(* CoDeSys 2.3 library: oscat152.lib *)
(* Libraries: Standard.lib 22.11.04 11:21:12 *)

(* Global variable list: Constants *)
VAR_GLOBAL CONSTANT
	(* Mathematische Konstanten *)
	PI : REAL := 3.14159265358979323846264338327950288;	(* Kreiszahl PI *)
	PI2 : REAL := 6.283185307179586476;							(* PI * 2 *)
	e : REAL := 2.71828182845904523536028747135266249;	(* Eulersche Konstante *)

	(* Physikalische Konstanten *)
	C0 : REAL := 299792458 ;										(* Lichtgeschwindigkeit in m/s *)
	EL : REAL := 1.60217653E-19;									(* elementarladung in Colomb = A * s *)
	GN : REAL := 9.80665; 											(* Erdbeschleunigung in m / s² *)
	TK : REAL := -273.15;												(* absoluter Nullpunkt in °C *)

END_VAR

VAR_GLOBAL
END_VAR

(* revisionhistory
hm 3.3.2007
	extended accuracy of pi2
	renamed T0 to Tk for better compatibility with other libraries
	renamed C t0 c0 for better compatibility
*)

(* Data type *)
TYPE esr_data :
STRUCT
	typ : BYTE;
	adress : STRING(10);
	DS : DT;
	TS : TIME;
	data : ARRAY[0..7] OF BYTE;
END_STRUCT
END_TYPE

(* POU _array_init, ST *)
FUNCTION _array_init : BOOL
VAR_INPUT
	pt : POINTER TO ARRAY[0..32000] OF REAL;
	size : INT;
	init : REAL;
END_VAR
VAR
	i: INT;
	stop: INT;
END_VAR


(*
version 1.1	9 jan 2007
programmer 	hugo
tested by		tobias

this function will initialize a given array with a value init.
the function needs to be called:	_array_init(adr("array"),sizeof("array"));
this function will manipulate a given array.
the function manipulates the original array, it rerturnes true when finished.
because this function works with pointers its very time efficient and it needs no extra memory.

*)
stop := (size - SIZEOF(pt)) / SIZEOF(pt);
FOR i := 0 TO stop DO
	pt^[i] := init;
END_FOR;
_array_init := TRUE;

(* revision History

hm 6.1.2007	rev 1.1
change typ of function to bool
added _array_init := true to set output true.

*)
END_FUNCTION

(* POU _array_median, ST *)
FUNCTION _array_median : REAL
VAR_INPUT
	pt : POINTER TO ARRAY[0..32000] OF REAL;
	size : INT;
END_VAR
VAR
	i: INT;
	m: INT;
	temp : REAL;
	stop: INT;
END_VAR

(*
version 1.1	3 mar 2007
programmer 	hugo
tested by		tobias

this function will calculate the median of a given array.
in order to do so the ariginal array is sorted and stays sorted after the function finishes
the function needs to be called:	_array_median(adr("array"),sizeof("array"));
this function will manipulate a given array.
the function will return the median of the original array.
for example [12,0,4,7,1] the median is 4 and the array after the function is called is [0,1,4,7,12]
because this function works with pointers its very time efficient and it needs no extra memory.

*)
stop := (size - SIZEOF(pt)) / SIZEOF(pt);
FOR i := 0 TO stop - 1 DO
	FOR m := i + 1 TO stop DO
		IF pt^[i] > pt^[m] THEN
			temp := pt^[i];
			pt^[i] := pt^[m];
			pt^[m] := temp;
		END_IF;
	END_FOR;
END_FOR;
IF even(stop) THEN
	_array_median := pt^[stop/2];
ELSE
	i := stop/2;
	_array_median := (pt^[i] + pt^[i+1])/2;
END_IF;

(* revision history
hm 3.3.2007	rev 1.1
	corrected an error, changed the statement line 14	i := TRUNC(stop/2); to i := stop/2;

*)
END_FUNCTION

(* POU even, ST *)
FUNCTION even : BOOL
VAR_INPUT
	in : INT;
END_VAR
VAR
END_VAR


(*
version 1.0	1 oct 2006
programmer 	hugo
tested by		tobias

this function chacks an input for even  value
the output is true if the input is even.
execution time on wago 750 - 841 =  10  us
*)
IF (in MOD 2) = 0 THEN  even := TRUE; ELSE even := FALSE; END_IF;
END_FUNCTION

(* POU _array_sort, ST *)
FUNCTION _array_sort : BOOL
VAR_INPUT
	pt : POINTER TO ARRAY[0..32000] OF REAL;
	size : INT;
END_VAR
VAR
	i: INT;
	m: INT;
	temp : REAL;
	stop: INT;
END_VAR

(*
version 1.1	6 jan 2007
programmer 	hugo
tested by		tobias

this function will sort a given array.
the function needs to be called:	_array_sort(adr("array"),sizeof("array"));
this function will manipulate a given array.
the function will not return anything except true, it will instead manipulate the original array.
because this function works with pointers its very time efficient and it needs no extra memory.

*)
stop := (size - SIZEOF(pt)) / SIZEOF(pt);
FOR i := 0 TO stop - 1 DO
	FOR m := i + 1 TO stop DO
		IF pt^[i] > pt^[m] THEN
			temp := pt^[i];
			pt^[i] := pt^[m];
			pt^[m] := temp;
		END_IF;
	END_FOR;
END_FOR;
_array_sort := TRUE;

(* revision history

hm 6.1.2007 	rev 1.1
	changed return value to true

*)
END_FUNCTION

(* POU acosH, ST *)
FUNCTION acosH : REAL
VAR_INPUT
	X : REAL;
END_VAR
VAR
END_VAR


(*
version 1.0	12 jan 2007
programmer 	hugo
tested by		tobias

this function calculates the arcus cos hyperbolicus

*)
acosH := LN(X + SQRT(EXPT(x,2)-1));
END_FUNCTION

(* POU acotH, ST *)
FUNCTION acotH : REAL
VAR_INPUT
	X : REAL;
END_VAR
VAR
END_VAR


(*
version 1.0	12 jan 2007
programmer 	hugo
tested by		tobias

this function calculates the arcus cotangens hyperbolicus

*)
acotH := LN((x+1)/(x-1))/2;
END_FUNCTION

(* POU actuator_2P, ST *)
FUNCTION_BLOCK actuator_2P
VAR_INPUT
	val : REAL;
	force : BOOL;
	force_in : BOOL;
END_VAR
VAR_INPUT CONSTANT
	self_act_time : TIME := t#10d;
	self_act_cycles : INT := 5;
	cycle_time : TIME := t#10m;
	min_ontime : TIME := t#10s;
	min_offtime : TIME := t#10s;
END_VAR
VAR_OUTPUT
	out :BOOL;
	pos : REAL;
END_VAR
VAR
	last_activation : TIME;
	count : INT;
	TON : TIME;
END_VAR


(*
version 1.2	17 jan 2007
programmer 	hugo
tested by		tobias

this is an intelligent actuator interface for any 2point actuator like coil drive.
the 2Point actuator can only switch on/off and therefore a input must be converted to on/off cycles.
the interface can be programmed with double click on the symbol for duty cyle, min_ontime and min_offtime to avoid flickering of the valve or flap.
in addition a self_act_time and self_act_cycles ca be programmed to switch n times on/off every self_act_time to avoid a valve to freeze.
a on and off input can be used to force the valve on or off at all times.
a additional pos output will always indicate the current position of a valve.
the input value must be between 0 and 1.

val		force	force_in	pos	out			
X		0		-			X		duty cycle X
-		1		1			1		1
-		1		0			0		0

*)
(* verify input to be between 0 and 1 *)
IF val <0 THEN val := 0; ELSIF val > 1 THEN val := 1; END_IF;

(* check for min ontime or min offtime and wait if not passed *)
IF (out AND TIME() - last_activation < min_ontime) OR (NOT out AND TIME() - last_activation < min_offtime) THEN RETURN;

(* when force off then shutoff valve *)
ELSIF force AND NOT force_in THEN
	pos := 0;
	out := 0;
	last_activation := TIME();
	count := 0;

(* if force on then turn on valve *)

ELSIF force AND force_in THEN
	pos := 1;
	out := 1;
	last_activation := TIME();
	count := 0;

(* if nothing happened for self_act_time then do self activation cycles *)
ELSIF (TIME() - last_activation >= self_act_time AND count = 0 AND self_act_cycles > 0) OR (count > 0 AND count < self_act_cycles * 2) THEN
	out := NOT out;
	last_activation := TIME();
	count := count + 1;
	RETURN;
ELSIF count > 0 THEN
	count := 0;
ELSE
	ton := multime(cycle_time,val);
	IF ton < min_ontime / 2 THEN ton := t#0s; ELSIF ton < min_ontime THEN ton := min_ontime; END_IF;
	IF ton > cycle_time - min_offtime / 2 THEN ton := cycle_time; ELSIF ton > cycle_time - min_offtime THEN ton := cycle_time - min_offtime; END_IF;
	IF ton = t#0s THEN
		IF out =0 THEN
			pos := 0;
			RETURN;
		ELSE
			out := 0;
			pos := 0;
			last_activation := TIME();
		END_IF;
	ELSIF ton = cycle_time THEN
		IF out = 1 THEN
			pos := 1;
			RETURN;
		ELSE
			out := 1;
			pos := 1;
			last_activation := TIME();
		END_IF;
	END_IF;
	pos := TIME_TO_REAL(ton) / TIME_TO_REAL(cycle_time);
	(* output pulse generation *)
	IF out AND TIME() - last_activation >= ton THEN
		out := 0;
		last_activation := TIME();
	ELSIF NOT out AND TIME() - last_activation >= cycle_time - ton THEN
		out := 1;
		last_activation := TIME();
	END_IF;
END_IF;


(*
revision history:

7.10.2006: rev 1.1
	changed error pos could not reach 1 or 0 under certain conditions due to error in code.
	changes on and off in the be force and force_in for better usability.

17.1.2007	rev 1.2
	deleted unused variable time_overflow
*)
END_FUNCTION_BLOCK

(* POU cycle_time, ST *)
FUNCTION_BLOCK cycle_time
VAR_INPUT
	rst : BOOL;
END_VAR
VAR_OUTPUT
	ct_min : TIME := t#0s;
	ct_max : TIME := t#0s;
	ct_last : TIME;
	systime : TIME;
	sysdays : INT;
	cycles : DWORD;
END_VAR
VAR
	last_cycle : TIME;
	tx: TIME;
	init: BOOL;
END_VAR


(*
	version 1.2	10 Mar 2007
	programmer 	hugo
	tested BY		hans

this function block measures the cycle time and displays the last, min and max cycle time of the current task.
the resolution is 1ms.
the cycles output is a dword counter which counts the cycles.
a rst pulse on the input will reset all data.


*)
tx :=TIME() - last_cycle;
IF rst THEN
	ct_min := t#10h;
	ct_max := t#0ms;
	cycles := 0;
ELSIF last_cycle > t#0s THEN
	IF tx < ct_min THEN ct_min := tx;
	ELSIF tx > ct_max THEN ct_max := tx;
	END_IF;
	ct_last := tx;
ELSIF ct_min = t#0s THEN
	ct_min := t#0s - t#1ms;
END_IF;
IF init THEN
	systime := systime + tx;
		IF systime >= t#1d THEN
			systime := systime - t#1d;
			sysdays := sysdays + 1;
		END_IF;
END_IF;
init := TRUE;
last_cycle := last_cycle + tx;
cycles := cycles + 1;

(*	revision history
hm 12.12.2006		rev 1.1
	added cycles output, a dword cycle counter.
hm 10.3.2007			rev 1.2
	changed initialization of ct_min to t#10h for compatibility with siemens s7

*)
END_FUNCTION_BLOCK

(* POU multime, ST *)
FUNCTION multime : TIME
VAR_INPUT
	t : TIME;
	M : REAL;
END_VAR
VAR
END_VAR


(*
version 1.0	2 oct 2006
programmer 	hugo
tested by		tobias

multiplies a time by a real number and returns a time
*)
multime := REAL_TO_TIME(TIME_TO_REAL(t)*M);
END_FUNCTION

(* POU actuator_3P, ST *)
FUNCTION_BLOCK actuator_3P
VAR_INPUT
	in : REAL;
	force : BOOL;
	on : BOOL;
	end_pos : BOOL;
	diag : BOOL;
END_VAR
VAR_INPUT CONSTANT
	min_ontime : TIME := t#10s;
	min_offtime : TIME := t#10s;
	max_runtime : TIME := t#60s;
	auto_diag_time : TIME := t#10d;
	cal_runtime : TIME := t#600s;
	switch_available: BOOL;
END_VAR
VAR_OUTPUT
	out1 : BOOL;
	out2 : BOOL;
	pos : REAL;
	busy : BOOL;
	error : BOOL;
END_VAR
VAR
	val: REAL;
	tx : TIME;
	last_diag: TIME;
	last : TIME;
	runtime_1 : TIME;
	runtime_2 : TIME;
	state : INT;
	rout: FT_rmp;
	end : R_TRIG;
	cal_timer: TIME;
END_VAR


(*
version 1.2	23 Jan 2007
programmer 	hugo
tested by		tobias

actuator_3P is an interface for a 3 point actuator.
a 3P actuator is a motor with 2 directions that drives a valve or flap. the position of the valve or flap is controlled by runtime of the motor foreward or backward.
the available inputs are:
in is a real value which specifies the position of the actuator, 0 = 0% and 1 = 100% any value <0 or > 1 is limited to 0 or 1.
a force input must be low for normal operation and if switched high, the motor can only be controlled for 0% or 100% positions with the on input.
an and pos input is available for a end_pos switch, this switch indicates the valve or flap to be at either 0% or 100%
a diag input can at any time start a diag cycle which turns the motor towards the 0% position, then measures the runtime to 100% and then the runtime to 0%
these runtimes are stored and used for absolute positioning of the motor during normal operation.
a setup constand "auto_diag_time can be used to specify how often the actuator repeates this auto_diag cycla automatically.
at power on a cycle is perfomed automatically.
a 0 for this value means auto diag is never performed.

the outputs ar out1 and out2 for up and down direction of the motor. to avoid flickering the output can be programmed for min_ontime and min_offtime.
a pos outout indicates the absulute position of the actuator during operation and a busy output indicates the actuator is busy.
a error output is initiated when the specified max_runtime is reached by any direction during debug.
also when the up and down direction differs by more then 10% the error output is set.

for absolute positioning accuracy the actuator has a setup variable "cal_runtime" if this is set the actuator measures the total runtime of the motors and when this 
cal_runtime is exceeded it resets the actuator to 0% position and sets the output again to assure absolute accuracy.

autodiag and calibration can be shut off by setting the appropriate values to 0.
a switch_available setup variable specifies if end_pos switches are available.

*)
(* setup *)
tx := TIME() - last;
end(clk := end_pos);

(* init only when first started *)
IF state = 0 THEN
	runtime_1 := max_runtime;
	runtime_2 := max_runtime;
	state := 1;
	rout(KR := 1000 / TIME_TO_REAL(runtime_1), KF := 1000 / TIME_TO_REAL(runtime_1) );
	tx := t#0s;
	last := TIME();
	last_diag := last;
END_IF;

(* check for end_sw and stop if reached *)
IF switch_available AND out1 AND end.Q THEN
	(* upper limit has been reached *)
	out1 := 0;
	rout(rmp := 0, in := 1);
	rout.Rmp := 1;
ELSIF switch_available AND out2 AND end.Q THEN
	(* lower limit has been reached *)
	out2 := 0;
	rout(rmp := 0, in := 0);
	rout.Rmp := 1;
END_IF;

(* check for min_offtime and min_ontime and return if it has not elapsed *)
IF NOT busy AND tx < min_offtime THEN RETURN;
ELSIF busy AND tx < min_ontime THEN RETURN;

(* check for last diag cycle and start diag if auto_diag_time has elapsed *)
ELSIF (tx + last - last_diag > auto_diag_time AND state > 10 AND auto_diag_time > t#0s) OR (diag AND state >= 10) THEN state := 1;

(* check if force pin is high *)
ELSIF force THEN state := 10;

(* check if calibration is necessary *)
ELSIF cal_timer > cal_runtime AND state = 99 AND cal_runtime > t#0s THEN state := 20;
END_IF;

(* state machine for operation *)
CASE state OF

1 :	(* diagnostic start *)
	(* all data is reset and out2 is turned on to make sure we start from top position *)
	last_diag := tx + last;
	diag := 0;
	state := 2;
	pos := 0;
	busy := 1;
	last := tx + last;
	out1 := 0;
	out2 := 1;
	RETURN;

2:	(* wait for max_runtime or end_pos to be reached *)
	IF tx < max_runtime AND NOT end.Q THEN RETURN; END_IF;
	state := 3;
	last := tx + last;
	out1 := 1;
	out2 := 0;
	RETURN;

3: 	(* measure runtime_2 *)
	IF tx < max_runtime AND NOT end.Q THEN RETURN; END_IF;
	state := 4;
	runtime_1 := tx;
	last := tx + last;
	out1 := 0;
	out2 := 1;
	RETURN;

4:	(* measure runtime_1 *)
	IF tx < max_runtime AND NOT end.Q THEN RETURN; END_IF;
	state := 99;
	runtime_2 := tx;
	last := tx + last;
	out2 := 0;
	busy := 0;
	(* reset the output ramp generator to the 0% position as the valve is after diags *)
	rout(rmp := 0, in := 0);
	rout.Rmp := 1;
	cal_timer := t#0s;
	IF differ(TIME_TO_REAL(runtime_1), TIME_TO_REAL(runtime_2), TIME_TO_REAL(max_runtime) * 0.1) THEN error := TRUE;
	ELSIF runtime_1 > multime(max_runtime, 0.9) AND switch_available THEN error := TRUE;
	ELSIF runtime_2 > multime(max_runtime, 0.9) AND switch_available THEN error := TRUE;
	END_IF;
	RETURN;

10: (* force pin is active, outputs are forced on or off by the on pin *)
	IF on AND NOT out2 THEN val := 1;
	ELSIF NOT on AND NOT out1 THEN val := 0;
	END_IF;
	IF NOT force THEN state := 99; END_IF;

20 : (* calibrate to allow for correction of positioning error addig up *)
	cal_timer := t#0s;
	state := 21;
	pos := 0;
	busy := 1;
	last := tx + last;
	out1 := 0;
	out2 := 1;
	RETURN;

21:	(* after end_sw or max_runtime we can be sure to have reached the 0% position *)
	IF tx < max_runtime AND NOT end.Q THEN RETURN; END_IF;
	state := 99;
	out2 := 0;
	busy := 0;
	last := tx + last;
	rout(rmp := 0, in := 0);
	rout.Rmp := 1;
	RETURN;

99: (* normal operation *)
	(* only if input changes for an equivalent of min_ontime then change the output *)
	(* if there is a directional change then wait until last step is finished *)
	IF in < TIME_TO_REAL(min_ontime)/TIME_TO_REAL(max_runtime)/2 THEN val := 0;
	ELSIF in > 1 - TIME_TO_REAL(min_ontime)/TIME_TO_REAL(max_runtime)/2 THEN val := 1;
	ELSIF differ(LIMIT(0,in,1), val, TIME_TO_REAL(min_ontime) / TIME_TO_REAL(max_runtime)) OR in = 0 OR in = 1 THEN
		IF in < val AND NOT out1 THEN val := in;
		ELSIF in > val AND NOT out2 THEN val := in;
		END_IF;
	END_IF;

END_CASE;

(* output ramp generator *)
rout(in := val);
out1 := rout.busy AND rout.UD;
out2 := rout.busy AND NOT rout.UD;
pos := rout.out;

(* set the busy output and if busy goes low, then set the last time in order to check for min_offtime *)
IF NOT busy AND rout.busy THEN
	last := tx + last;
ELSIF busy AND NOT rout.busy THEN
	cal_timer := cal_timer + tx;
	last := tx + last;
END_IF;
busy := rout.busy;



(* revision history

19.10.2006	rev 1.1
	added security checks for end_switch to avoid overrun of the end_switch, hans

23.1.2007		rev 1.2
	deleted unused variables force_on and force_off


*)
END_FUNCTION_BLOCK

(* POU FT_rmp, ST *)
FUNCTION_BLOCK FT_rmp
VAR_INPUT
	Rmp : BOOL := TRUE;
	in : REAL;
	KR : REAL;
	KF : REAL;
END_VAR
VAR_OUTPUT
	out : REAL;
	busy : BOOL;
	UD : BOOL;
END_VAR
VAR
	tx: TIME;
	last: TIME;
	init: BOOL;
END_VAR

(*
	version 1.2	12 Feb 2007
	programmer 	oscat
	tested BY		oscat

this ramp function follows an input signal with a linear ramp up or down, the up or down speed can be set with KF and KR.
a K factor of 1 means 1 unit per second on the output. K factors can only be positive and not negative.
a busy output signals the ramp is running or busy false means the in value is present on the output.
a rmp input false means the output follows the input dierctly while a rmp = true means the output follows the input with a ramp.
a updn output signal the directon of the ramp (up or down).

*)
tx := TIME() - last;
IF NOT init THEN
	init := TRUE;
	last := tx;
	tx := t#0s;
	out := in;
END_IF;
IF NOT rmp THEN
	out := in;
	busy := FALSE;
ELSIF out > in AND kf > 0 THEN
	(* ramp down *)
	out := out - TIME_TO_REAL(tx) / 1000 * KF;
	IF out < in THEN out := in; END_IF;
ELSIF out < in AND kr > 0 THEN
	(* ramp up *)
	out := out + TIME_TO_REAL(tx) / 1000 * KR;
	IF out > in THEN out := in; END_IF;
END_IF;

(* set busy and dir flags *)
IF out < in THEN
	busy := TRUE;
	ud := 1;
ELSIF out > in THEN
	busy := TRUE;
	ud := 0;
ELSE
	busy := FALSE;
END_IF;
last := last + tx;


(* revision history:

hm 8.10.2006			rev 1.1
	added ud output

hm 12. feb 2007		rev 1.12
	added init variable and corrected a possible startup problem
*)
END_FUNCTION_BLOCK

(* POU differ, ST *)
FUNCTION differ : BOOL
VAR_INPUT
	in1 : REAL;
	in2 : REAL;
	X : REAL;
END_VAR
VAR
END_VAR

(*
version 1.0	8 oct 2006
programmer 	hugo
tested by		tobias

this function checks if in1 differs more then x from in2
the output is true if in1 < in2 - x or in1 > in2 + X
*)
differ := in1 < in2 - X OR in1 > in2 + X;
END_FUNCTION

(* POU actuator_pump, ST *)
FUNCTION_BLOCK actuator_pump
VAR_INPUT
	in : BOOL;
	manual : BOOL;
	rst : BOOL := FALSE;
END_VAR
VAR_INPUT CONSTANT
	min_ontime : TIME := t#10s;
	min_offtime : TIME := t#10s;
	run_every : TIME := t#10000m;
END_VAR
VAR_OUTPUT
	pump : BOOL;
	runtime : REAL;
	cycles : REAL;
END_VAR
VAR
	tx : TIME;
	last_change : TIME;
	meter : ontime;
	old_man : BOOL;
	init: BOOL;
END_VAR

(*
	version 1.1	27 dec 2006
	programmer 	oscat
	tested BY		oscat

actuator_pump is a pump interface which can be controlled by an input in and an input manual.
in or manual high turns the pump output on.
a rst input is used to reset the runtime counters.
when the pump was not active for a time run_every the actuator turns on the pump automatically for min_ontime.
two setup variables min_ontime and min_offtime guarantee a minimum runtime and offtime of the pump.
the units are hours and the output type is real to prevent from overfow.

*)
tx := TIME();

IF NOT init THEN
	init := 1;
	last_change := tx;
ELSIF rst THEN
	rst := FALSE;
	meter(rst := 1);
	meter.rst := 0;
ELSIF manual AND NOT pump AND NOT old_man THEN
	last_change := tx;
	pump := 1;
ELSIF NOT manual AND old_man AND pump AND NOT in THEN
	last_change := tx;
	pump := 0;
ELSIF in AND NOT pump AND tx - last_change >= min_offtime THEN
	last_change := tx;
	pump := 1;
ELSIF pump AND NOT in AND NOT manual AND tx - last_change >= min_ontime THEN
	last_change := tx;
	pump := 0;
ELSIF NOT pump AND tx - last_change >= run_every THEN
	last_change := tx;
	pump := 1;
END_IF;

meter(in := pump);
runtime := meter.ontime;
cycles := meter.cycles;
old_man := manual;

(*
27.12.2006	rev 1.1	hm
fixed a failure while the pump would run for tmin after startup.


*)
END_FUNCTION_BLOCK

(* POU ontime, ST *)
FUNCTION_BLOCK ontime
VAR_INPUT
	in : BOOL;
	rst : BOOL := FALSE;
END_VAR
VAR_OUTPUT RETAIN
	ontime : REAL;
	last_on : REAL;
	cycles : REAL;
END_VAR
VAR
	tx: TIME;
	last : TIME;
	power : BOOL := FALSE;
	edge : BOOL := 0;
END_VAR

(*
version 1.1	22 feb 2007
programmer 	oscat
tested by		tobias

M_runtime measures the ontime of a signal in hours.
the output is of type real because the time type will overflow within 49 days.
the units are hours.

*)
(* at first we need to determine if the sps was powered off *)

tx := TIME();
IF NOT power THEN
	power := TRUE;
	cycles := cycles +1;
ELSIF rst THEN
	ontime := 0;
	cycles := 0;
	last_on := 0;
ELSIF in THEN
	ontime := ontime + DWORD_TO_REAL( TIME_TO_DWORD(tx - last))/3600000.0;
	last_on := last_on + DWORD_TO_REAL(TIME_TO_DWORD(tx - last))/3600000.0;
	IF in AND NOT edge THEN
		cycles := cycles +1;
		last_on := 0;
	END_IF;
END_IF;
last := tx;
edge := in;

(* revision history
hm 22.2.2007		rev 1.1
	changed VAR RETAIN PERSISTENT to VAR RETAIN for better compatibility
	wago lon contollers do not support persisitent

*)
END_FUNCTION_BLOCK

(* POU actuator_UD, ST *)
FUNCTION_BLOCK actuator_UD
VAR_INPUT
	UD : BOOL;
	ON : BOOL;
	Manual : BOOL := 0;
	Up : BOOL;
	Dn : BOOL;
	off : BOOL := 0;
	YUP_in : BOOL;
	YDN_in : BOOL;
END_VAR
VAR_INPUT CONSTANT
	TON : TIME;
	TOFF : TIME;
	out_return : BOOL;
END_VAR
VAR_OUTPUT
	Yup : BOOL;
	Ydn : BOOL;
	status : BYTE;
END_VAR
VAR
	tx : TIME;
	last : TIME;
	init: BOOL;
END_VAR

(*
version 1.1	22 jan 2007
programmer 	hugo
tested by		tobias

out_ud is a up/dn or Right/left locked output driver.
it can be controlled by automatic inputs UD and ON as well as manual inputs for up and dn.
a security input to shut off at any time is prvided by the off input.
two time set inputs ton and toff specify a minimum on time for outputs and a minimum off time before the next output can become active.
the module assures that only one output can be active at any time.
for higher security pls make sure you use hardware locking of the outputs to prevent from defective wiring or outputs.
further security is provided b feedback inputs Yup_in and Ydn_in which are separate inputs for the output signal, if these inputs are not available 
pls connect them directly to Yup and Ydn.
manual mode will override automatic mode by setting the manual input high.
a status output will be 0 for normal operation or 1 - 99 for error reporting and 101 - 199 for status reporting
The status output is ESR comptible.
*)
(* read system time *)
tx := TIME();

IF NOT init THEN
	(* INITIALIZATION AT FIRST CALL *)
	last := tx;
	init := TRUE;
ELSIF off THEN
	(* emergency shut off detected *)
	Yup := FALSE;
	Ydn := FALSE;
	last := tx;
	status := 101;

(* WATH FOR MIN TON TIME *)
ELSIF ((Yup OR Ydn) AND tx - last < Ton) THEN RETURN;
ELSIF NOT yup AND NOT ydn AND tx - last < toff THEN	RETURN;

(* manual operation *)
ELSIF manual THEN
	status := 102;
	(* directional chage set both outs 0 first *)
	IF yup AND NOT up OR ydn AND NOT dn THEN
		ydn := 0;
		yup := 0;
		last := tx;
	(* manual up operation *)
	ELSIF UP AND NOT DN AND NOT OFF THEN
		Ydn := 0;
		Yup := 1;
		last := tx;
		status := 103;
	(* manual down operation *)
	ELSIF DN AND NOT UP AND NOT OFF THEN
		Yup := 0;
		Ydn := 1;
		last := tx;
		status := 104;
	(* maual mode but no up or down *)
	ELSE
		IF YUP OR YDN THEN LAST := tx; END_IF;
		Yup := 0;
		Ydn := 0;
	END_IF;

(* automatic operation *)
ELSE
	(* directional change set outputs low first *)
	IF yup AND NOT ud OR ydn AND UD THEN
		yup := 0;
		ydn := 0;
		last := tx;
	(* automatic up operation *)
	ELSIF Ud AND on AND NOT OFF THEN
		Ydn := 0;
		Yup := 1;
		last := tx;
		status := 111;

	(* automatic down operation *)
	ELSIF NOT UD AND on AND NOT OFF THEN
		Yup := 0;
		Ydn := 1;
		last := tx;
		status := 112;
	(* standby mode *)
	ELSE
		IF Yup OR Ydn THEN last := tx; END_IF;
		Yup := 0;
		Ydn := 0;
		status := 110;
	END_IF;
END_IF;

(* make sure Yup and Ydn are never on at the same time *)
IF Ydn AND Yup_in AND out_return THEN
	Ydn := 0;
	status := 1;
END_IF;
IF Yup AND Ydn_in AND out_return THEN
	Yup := 0;
	status := 2;
END_IF;

(* revision history
hm 22. jan 2007	rev 1.1
	added status output
	changed inputs ton, toff to config variables
	added config var out_return to enable yup_in and Ydn_in
	manual mod will override automatic mode 
*)
END_FUNCTION_BLOCK

(* POU AIN, ST *)
FUNCTION AIN : REAL
VAR_INPUT
	in : DWORD;
END_VAR
VAR_INPUT CONSTANT
	Bits : BYTE;
	sign : BYTE := 255;
	low : REAL := 0;
	high : REAL := 10;
END_VAR
VAR
	temp1 : DWORD;
	temp2 : DWORD;
	sx : BOOL;
END_VAR

(*
version 1.2	19 jan 2007
programmer 	oscat
tested by		tobias

Ain converts signals from A/D converters or other analog sources to an internal real value
the lowest number of bits are extracted from the input word and the sign will be extracted if available separately.
the output signal is then conditioned to range from low to high values for a 0 to max value on the analog inputs:
for example a 15bit input (bits := 12) with sign at bit 15 (0..15) will deliver 0.0 (low value at 0) for an input value of 2#0000_0000_0000
an input value of 2#1111_1111_1111 will deliver 10.0 on the output (high value set to 10).

*) 
(* extract the sign bit *)
IF sign < 32 THEN
	temp1 := SHR(in,sign);
	sx := temp1.0;
ELSE
	sx := FALSE;
END_IF;
temp1 := SHR(16#FFFFFFFF,32-bits);
temp2 := in AND temp1;
AIN := (high - low)*temp2 / temp1 + low;
IF sx THEN AIN := AIN * -1; END_IF;

(* revision history
hm 18.8.2006	rev 1.1
	fixed an error with low value negative and high value 0.

hm 19.1.2007	rev 1.2
	fixed an error with sign bit.
*)
END_FUNCTION

(* POU Aout, ST *)
FUNCTION Aout : DWORD
VAR_INPUT
	in : REAL;
END_VAR
VAR_INPUT CONSTANT
	Bits : BYTE;
	sign : BYTE := 255;
	low : REAL := 0;
	high : REAL := 10;
END_VAR
VAR
	in2 : REAL;
	sx : BOOL;
END_VAR

(*
version 1.1	18 jan 2007
programmer 	oscat
tested by		tobias

this module conditions an internal real value for a signal output D/A converter.
Aout converts and internal real value to a word for an D/A converter or other output devices.
The input value is converted to a n-bit wide output and a sign bit is set separately as specified.
the outout min value is set for the specified min input value and the max output is set for the max input value.
an input higher or lower then the max or min value will set the respective max or min value or the output.


*) 
(* if sign bit is defined *)
IF sign < 32 THEN
	sx := sign_R(in);
	in2 := ABS(in);
ELSE
	in2 := in;
END_IF;

(* begrenze in auf die zulässigen werte *)
IF in2 < low THEN
	in2 := low;
ELSIF in2 > high THEN
	in2 := high;
END_IF;

(* Berechne den Ausgnagswert *)
Aout := REAL_TO_DWORD((in2 - low) / (high - low) * (EXPT(2,bits) -1));
IF sx THEN Aout := SHL(2#1,sign) OR Aout; END_IF;

(*
revision history

hm 17.1.2007		rev 1.1
	renamed Modul to aout.
	changed Output to 32 Bit max.
	corrected error with sign bit.
*)
END_FUNCTION

(* POU sign_R, ST *)
FUNCTION sign_R : BOOL
VAR_INPUT
	in : REAL;
END_VAR
VAR
END_VAR

(*
version 1.1	19 jan 2007
programmer 	hugo
tested by		tobias

this function return true if the real input is negative

*)
IF in < 0 THEN
	sign_R := TRUE;
ELSE
	sign_R := FALSE;
END_IF;

(* revision history
hm 19.1.2007	rev 1.1
	changed method of function for better compatibility to other systems

*)
END_FUNCTION

(* POU array_avg, ST *)
FUNCTION array_avg : REAL
VAR_INPUT
	pt : POINTER TO ARRAY[0..32000] OF REAL;
	size : INT;
END_VAR
VAR
	i: INT;
	stop: INT;
END_VAR

(*
version 1.0	2 oct 2006
programmer 	hugo
tested by		tobias

this function will calculate the average of a given array.
the function needs to be called:	array_avg(adr("array"),sizeof("array"));
because this function works with pointers its very time efficient and it needs no extra memory.

*)
stop := (size -SIZEOF(pt)) / SIZEOF(pt);
array_avg := pt^[0];
FOR i := 1 TO stop DO
	array_avg := array_avg + pt^[i];
END_FOR;
array_avg := array_avg / (stop + 1);
END_FUNCTION

(* POU array_max, ST *)
FUNCTION array_max : REAL
VAR_INPUT
	pt : POINTER TO ARRAY[0..32000] OF REAL;
	size : INT;
END_VAR
VAR
	i: INT;
	stop: INT;
END_VAR

(*
version 1.0	2 oct 2006
programmer 	hugo
tested by		tobias

this function will calculate the max value of a given array.
the function needs to be called:	array_max(adr("array"),sizeof("array"));
because this function works with pointers its very time efficient and it needs no extra memory.

*)
stop := (size -SIZEOF(pt)) / SIZEOF(pt);
array_max := pt^[0];
FOR i := 1 TO stop DO
	IF pt^[i] > array_max THEN array_max := pt^[i]; END_IF;
END_FOR;
END_FUNCTION

(* POU array_min, ST *)
FUNCTION array_min : REAL
VAR_INPUT
	pt : POINTER TO ARRAY[0..32000] OF REAL;
	size : INT;
END_VAR
VAR
	i: INT;
	stop: INT;
END_VAR

(*
version 1.0	2 oct 2006
programmer 	hugo
tested by		tobias

this function will calculate the min value of a given array.
the function needs to be called:	array_min(adr("array"),sizeof("array"));
because this function works with pointers its very time efficient and it needs no extra memory.

*)
stop := (size - SIZEOF(pt)) / SIZEOF(pt);
array_min := pt^[0];
FOR i := 1 TO stop DO
	IF pt^[i] < array_min THEN array_min := pt^[i]; END_IF;
END_FOR;
END_FUNCTION

(* POU array_spr, ST *)
FUNCTION array_spr : REAL
VAR_INPUT
	pt : POINTER TO ARRAY[0..32000] OF REAL;
	size : INT;
END_VAR
VAR
	i: INT;
	stop: INT;
	array_max : REAL;
	array_min : REAL;
END_VAR

(*
version 1.0	2 oct 2006
programmer 	hugo
tested by		tobias

this function will calculate the spread of a given array.
the function needs to be called:	array_spr(adr("array"),sizeof("array"));
for example: spread of [12,0,4,1,7] is 12 - 0 = 12.
because this function works with pointers its very time efficient and it needs no extra memory.

*)
stop := (size -SIZEOF(pt)) / SIZEOF(pt);
array_min := pt^[0];
array_max := pt^[0];
FOR i := 1 TO stop DO
	IF pt^[i] > array_max THEN array_max := pt^[i];
	ELSIF pt^[i] < array_min THEN array_min := pt^[i];
	END_IF;
END_FOR;
array_spr := array_max - array_min;
END_FUNCTION

(* POU array_sum, ST *)
FUNCTION array_sum : REAL
VAR_INPUT
	pt : POINTER TO ARRAY[0..32000] OF REAL;
	size : INT;
END_VAR
VAR
	i: INT;
	stop: INT;
END_VAR


(*
version 1.0	2 oct 2006
programmer 	hugo
tested by		tobias

this function will calculate the sum of a given array.
the function needs to be called:	array_sum(adr("array"),sizeof("array"));
because this function works with pointers its very time efficient and it needs no extra memory.

*)
stop := (size -SIZEOF(pt)) / SIZEOF(pt);
array_sum := pt^[0];
FOR i := 1 TO stop DO
	array_sum := array_sum + pt^[i];
END_FOR;
END_FUNCTION

(* POU array_trend, ST *)
FUNCTION array_trend : REAL
VAR_INPUT
	pt : POINTER TO ARRAY[0..32000] OF REAL;
	size : INT;
END_VAR
VAR
	i: INT;
	stop: INT;
	x: REAL;
	y : REAL;
END_VAR

(*
version 1.0	2 oct 2006
programmer 	hugo
tested by		tobias

this function will calculate the trend of a given array.
trend will calculate the avg of the first half of the array and then the avg of the second half, trend = avg2 - avg1.
for example:  [0,1,4,5,3,4,6,3] = 4 - 2.5 = 1.5
the function needs to be called:	array_trend(adr("array"),sizeof("array"));
because this function works with pointers its very time efficient and it needs no extra memory.

*)
stop := (size - SIZEOF(pt)) / SIZEOF(pt);
FOR i := 0 TO stop / 2 DO x := x + pt^[i]; END_FOR;
X := x / (TRUNC(stop / 2) + 1);
IF even(stop) THEN
	FOR i := stop / 2 TO stop DO y := y + pt^[i]; END_FOR;
	y := y / (stop / 2 + 1);
ELSE
	FOR i := TRUNC(stop / 2) + 1 TO stop DO y := y + pt^[i]; END_FOR;
	y := y / (TRUNC(stop / 2) + 1);
END_IF;
array_trend := y - x;
END_FUNCTION

(* POU asinH, ST *)
FUNCTION asinH : REAL
VAR_INPUT
	X : REAL;
END_VAR
VAR
END_VAR


(*
version 1.0	12 jan 2007
programmer 	hugo
tested by		tobias

this function calculates the arcus sin hyperbolicus

*)
asinH := LN(X + SQRT(EXPT(x,2)+1));
END_FUNCTION

(* POU atanH, ST *)
FUNCTION atanH : REAL
VAR_INPUT
	X : REAL;
END_VAR
VAR
END_VAR


(*
version 1.0	12 jan 2007
programmer 	hugo
tested by		tobias

this function calculates the arcus tangens hyperbolicus

*)
atanH := LN((1+x)/(1-x)) / 2;
END_FUNCTION

(* POU B_TRIG, ST *)
FUNCTION_BLOCK B_TRIG
VAR_INPUT
	CLK : BOOL;
END_VAR
VAR_OUTPUT
	Q : BOOL := 0;
END_VAR
VAR
	edge : BOOL := 0;
END_VAR

(*
version 1.0	4 aug 2006
programmer 	hugo
tested by		tobias

this block is similar to R_trig and F_trig but it generates a pulse on rising and falling edge.

executioin TIME on wago 750-841 = 5us
*)
Q := clk XOR edge;
edge := CLK;
END_FUNCTION_BLOCK

(* POU bar_graph, ST *)
FUNCTION_BLOCK bar_graph
VAR_INPUT
	X : REAL;
	rst : BOOL;
END_VAR
VAR_INPUT CONSTANT
	trigger_Low : REAL;
	trigger_High : REAL;
	Alarm_low : BOOL;
	Alarm_high : BOOL;
	log_scale : BOOL;
END_VAR
VAR_OUTPUT
	LOW, Q1, Q2, Q3, Q4, Q5, Q6, HIGH : BOOL;
	Alarm : BOOL;
	Status : BYTE;
END_VAR
VAR
	init : BOOL;
	T1, T2, T3, T4, T5 : REAL;
END_VAR
VAR_TEMP
	temp : REAL;
END_VAR
IF NOT init THEN
	init := TRUE;
	IF log_scale THEN
		temp := EXPT(Trigger_high / Trigger_low, 1 / 6);
		T1 := trigger_low * temp;
		T2 := T1 * temp;
		T3 := T2 * temp;
		T4 := T3 * temp;
		T5 := T4 * temp;
	ELSE
		temp := (trigger_high - trigger_low) / 7;
		T1 := trigger_low + temp;
		T2 := T1 + temp;
		T3 := T2 + temp;
		T4 := T3 + temp;
		T5 := T4 + temp;
	END_IF;
END_IF;

(* clear outputs before checking *)
Q1 := FALSE;
Q2 := FALSE;
Q3 := FALSE;
Q4 := FALSE;
Q5 := FALSE;
Q6 := FALSE;
status := 110;

(* low, high and alarm can only be cleared with rst depending on alarm_low and alarm_high *)
IF NOT alarm_low THEN low := FALSE; END_IF;
IF NOT alarm_high THEN high := FALSE; END_IF;
IF rst THEN
	alarm := FALSE;
	low := FALSE;
	high := FALSE;
END_IF;

(* check and set outputs *)
IF X < trigger_low THEN
	Low := TRUE;
	status := 111;
	IF alarm_low THEN
		alarm := TRUE;
		status := 1;
	END_IF;
ELSIF X < T1 THEN
	Q1 := TRUE;
ELSIF x < t2 THEN
	Q2 := TRUE;
ELSIF x < t3 THEN
	Q3 := TRUE;
ELSIF x < T4 THEN
	Q4 := TRUE;
ELSIF x < T5 THEN
	q5 := TRUE;
ELSIF x < trigger_high THEN
	q6 := TRUE;
ELSE
	high := TRUE;
	status := 112;
	IF alarm_high THEN
		alarm := TRUE;
		status := 2;
	END_IF;
END_IF;
END_FUNCTION_BLOCK

(* POU Bit_of_Dword, ST *)
FUNCTION Bit_of_Dword : BOOL
VAR_INPUT
	in : DWORD;
	N : BYTE;
END_VAR
VAR
	temp: DWORD;
END_VAR

(*
version 1.0	4 aug 2006
programmer 	hugo
tested by		tobias

this function extracts a single bit from the nth position from right (right is lowest bit)
the lowest Bit (Bit0 from in) is selected with N=0.
 *)
temp := SHR(in,n);
Bit_of_Dword := temp.0;
END_FUNCTION

(* POU Boiler, ST *)
FUNCTION_BLOCK Boiler
VAR_INPUT
	T_upper : REAL;
	T_lower : REAL;
	Pressure : BOOL := TRUE;
	enable : BOOL := TRUE;
	Req_1 : BOOL;
	Req_2 : BOOL;
	Boost : BOOL;
END_VAR
VAR_INPUT CONSTANT
	t_upper_min : REAL := 50;
	t_upper_max : REAL := 60;
	T_lower_enable : BOOL;
	T_lower_max : REAL := 60;
	T_request_1 : REAL := 70;
	T_request_2 : REAL := 50;
	T_request_hys : REAL := 5;
	T_protect_high : REAL := 80;
	T_protect_low : REAL := 10;
END_VAR
VAR_OUTPUT
	Heat : BOOL;
	error : BOOL;
	status : BYTE;
END_VAR
VAR
	edge: BOOL;
	boost_mode: BOOL;
	flag_0 : BOOL;
	flag_1: BOOL;
	flag_2: BOOL;
END_VAR

(*
version 1.0	27 feb 2007
programmer 	hugo
tested by		tobias

this function block controls a hot water boiler. The Boiler can be equipped with two temperature sensors on top and bottom of the tank, T_LOWER_ENABLE must be set to True in this case.
alternatively can BOILER be configured for one (TOP) temperature sensor only (T_LOWER_ENABLE set to False).
A Pressure sensor is used to detect fresh water pressure and disable all heating if there is no water pressure. This input is dset to True by default, so if it is not used it can simply be left open.
A enable input enables the hot water heating while it is set to True. alternatively can a Ture on Req_1 or Req_2 start the heating to predefined temperatures during setup.
A low to high edge on the boost input will start heating imediately until T_upper_max is reached, it can be used to generate extra hot water when needed.

*)
(* read sensors and check for valid data *)
IF t_upper > t_protect_high THEN
	status := 1;
	heat := FALSE;
	error := TRUE;
ELSIF t_upper < t_protect_low THEN
	status := 2;
	heat := TRUE;
	error := TRUE;
ELSIF t_lower > T_protect_high AND t_lower_enable THEN
	status := 3;
	heat := FALSE;
	error := TRUE;
ELSIF t_lower < t_protect_low AND t_lower_enable THEN
	status := 4;
	heat := TRUE;
	error := TRUE;
ELSIF NOT pressure THEN
	status := 5;
	heat := FALSE;
	error := TRUE;
ELSIF req_1 OR req_2 OR enable OR boost THEN
	error := FALSE;

	(* determine if heat needs to be turned on *)
	IF boost AND NOT edge AND t_upper < t_upper_max THEN
		status := 101;
		heat := TRUE;
		boost_mode := TRUE;
	ELSIF enable AND t_upper < T_upper_min THEN
		status := 102;
		heat := TRUE;
	ELSIF req_1 AND t_upper < T_request_1 THEN
		status := 103;
		heat := TRUE;
	ELSIF req_2 AND t_upper < t_request_2 THEN
		status := 104;
		heat := TRUE;
	END_IF;

	(* determine the shut off temperature *)
	IF heat THEN
		IF (enable OR boost_mode) THEN
			flag_0 := TRUE;
			IF T_lower_enable AND T_lower > T_lower_max THEN
				flag_0 := FALSE;
				boost_mode := FALSE;
			ELSIF NOT T_lower_enable AND T_upper > T_upper_max THEN
				flag_0 := FALSE;
				boost_mode := FALSE;
			END_IF;
		ELSE
			flag_0 := FALSE;
		END_IF;
		IF req_1 AND T_upper > T_request_1 + T_request_hys THEN flag_1 := FALSE; ELSE flag_1 := req_1; END_IF;
		IF req_2 AND T_upper > T_request_2 + T_request_hys THEN flag_2 := FALSE; ELSE flag_2 := req_2; END_IF;

		(* shut off heat if no longer needed *)
		heat := flag_0 OR flag_1 OR flag_2;
		IF heat = FALSE THEN status := 100; END_IF;
	END_IF;
ELSE
	status := 100;
	heat := FALSE;
	error := FALSE;
END_IF;
edge := boost;
END_FUNCTION_BLOCK

(* POU Burner, ST *)
FUNCTION_BLOCK Burner
VAR_INPUT
	in : BOOL;
	stage2 : BOOL;
	over_temp : BOOL;
	oil_temp : BOOL := TRUE;
	Flame : BOOL;
	rst : BOOL;
	rst_timer : BOOL;
END_VAR
VAR_INPUT CONSTANT
	pre_heat_time : TIME := t#5s;
	pre_vent_time : TIME := t#15s;
	pre_ignite_time : TIME := t#5s;
	post_ignite_time : TIME := t#25s;
	stage2_delay : TIME := t#10s;
	safety_time : TIME := t#5s;
	lockout_time : TIME := t#10s;
	multiple_ignition : BOOL := TRUE;
	KW1 : REAL;
	KW2 : REAL;
END_VAR
VAR_OUTPUT
	motor : BOOL;
	coil1 : BOOL;
	coil2 : BOOL;
	pre_heat: BOOL;
	ignite : BOOL;
	runtime1 : REAL;
	runtime2 : REAL;
	KWh : REAL;
	cycles : REAL;
	status : BYTE;
	fail : BOOL;
END_VAR
VAR
	state : BYTE;
	last : TIME;
	tx: TIME;
	last_change: TIME;
	timer1 : ontime;
	timer2 : ontime;
	oil_temp_last: BOOL;
END_VAR

(*
version 1.4	22 jan 2006
programmer 	oscat
tested by		tobias

burner ist eine Oel-Brenner_steuerung fuer nichtmodulierende Oelbrenner
die steuerung kann ueber setup werte programmiert werden und entsprechenden brennern angepasst werden.
die vorheizzeit ist die zeit die eine oelvorwaermung aufgeheizt wird bevor der motor gestartet wird.
der eingang oil_temp gibt an ob die oil_temp erreicht wurde, er ist default auf true und kann auch offen gelassen werden.
die vorbelueftungszeit ist die zeit die der luefter laeuft bevor die oelzufuhr freigegeben wird.
die vorzuendzeit iust diejenige zeit die die zuendung vor offnen des oelventiel gestartet wird.
nachzuendzeit ist die zeit die nach entzuendung der flamme noch gezuendet wird.
die sicherheitszeit ist die zeit nach der die oelzufuhr gesperrt wird wenn keine flamme entsteht.
nach ablauf der sicherheitszeit wird ein fehler flag gesetzt und kann erst nach der sperrzeit wieder durch einen reset geloescht werden.
waehrend der sperrzeit ist keine weitere zuendung oder einschalten moeglich.
das flag mehrfachzuendung gibt an ob eine erloschene flamme in betrieb automatisch wieder gezuendet werden soll.
der flammwaechster liegt auf eingang flamme, ein uebertemperaturschutz auf dem eingang over_temp
der betriebsstundenzaehler gibt die brennerstunden in stunden als real ausgabewer an.
der ausgang motor steuert den luefter / pumpenmotor, oil_ventil schaltet das oil ventil und zuendung schaltet die zuendung ein.

if output fail > 0 an error happened and the output has an error code:
0 :	no error
1 :	pre heating time expired and oil temp input is not true
2 :	flame monitor is active during preheating time
3 :	flame monitor active during pre_ventilation_time
4 :	no ignoition during safety time
5 :	no flame during operation
9 :	overtemp input is true

*)
tx := TIME();

(* check rst input and overtemp *)
IF rst OR over_temp OR state = 0 THEN
	IF status > 0 AND tx - last_change >= lockout_time AND rst THEN
		status := 110;
		fail := FALSE;
		state := 1;
	ELSE
		(* normaler reset *)
		motor := FALSE;
		coil1 := FALSE;
		coil2 := FALSE;
		ignite := FALSE;
		pre_heat := FALSE;
		IF over_temp THEN
			status := 9;
			fail := TRUE;
		END_IF;
		last_change := tx;
		last := tx;
		state := 1;
	END_IF;
END_IF;

(* check for timer rst and rst timer if true *)
IF rst_timer THEN
	timer1( rst := TRUE);
	timer1.rst := FALSE;
	timer2(rst := TRUE);
	timer2.rst := FALSE;
END_IF;

(* quit here if an error is present *)
IF (status > 0 AND status < 100) OR rst THEN RETURN; END_IF;

(* start sequence *)
CASE state OF

1:	(* in signal starts oil pre heating *)
	IF in AND flame THEN
		state := 7;
		pre_heat := FALSE;
		status := 2;
		last_change := tx;
	ELSIF in THEN
		pre_heat := TRUE;
		state := 2;
		last_change := tx;
	END_IF;

2:	(* after pre_heating time start motor *)
	IF (tx- last_change >= pre_heat_time AND oil_temp) OR (oil_temp AND NOT oil_temp_last) THEN
		motor := TRUE;
		state := 3;
		last_change := tx;
	(* pre_heat_time ist abgelaufen und oil_temp ist nicht aktiv *)
	ELSIF tx - last_change >= pre_heat_time AND NOT oil_temp THEN
		state := 7;
		pre_heat := FALSE;
		status := 1;
		last_change := tx;
	(* flame monitor cannot be active at this time *)
	ELSIF flame THEN
		state := 7;
		pre_heat := FALSE;
		status := 2;
		last_change := tx;
	END_IF;

3:	(* abwarten bis zündung eingeschaltet werden kann *)
	IF tx - last_change >= pre_vent_time - pre_ignite_time THEN
		ignite := TRUE;
		state := 4;
		last_change := tx;
	(* flame monitor cannot be active at this time *)
	ELSIF flame THEN
		state := 7;
		pre_heat := FALSE;
		motor := FALSE;
		status := 3;
		last_change := tx;
	END_IF;

4:	(* warten bis oelzufuhr geoeffnet werden darf *)
	IF tx - last_change >= pre_ignite_time THEN
		coil1 := TRUE;
		state := 5;
		last_change := tx;
	END_IF;

5:	(* warten auf flammwaechter und falls noetig abschalten *)
	IF tx - last_change >= safety_time OR flame THEN
		IF NOT flame THEN
			(* notabschaltung da flammwaechster nicht angesprochen hat *)
			state := 7;
			motor := FALSE;
			coil1 := FALSE;
			pre_heat := FALSE;
			ignite := FALSE;
			status := 4;
			last_change := tx;
		ELSE
			state := 6;
			last_change := tx;
		END_IF;
	END_IF;

6:	(* brenner läuft, flammueberwachung und nach ablauf der nachigniteszeit ignite abschalten *)
	IF NOT flame AND NOT multiple_ignition THEN
		(* notabschaltung da flammwaechster keine flamme meldet *)
		state := 7;
		motor := FALSE;
		coil1 := FALSE;
		coil2 := FALSE;
		pre_heat := FALSE;
		ignite := FALSE;
		status := 5;
		last_change := tx;
	ELSIF NOT flame AND multiple_ignition THEN
		ignite := TRUE;
		state := 5;
		coil2 := FALSE;
		last_change := tx;
	ELSE
		IF tx - last_change >= post_ignite_time THEN
			(* post_ignite_time abgelaufen, ignite abschalten *)
			ignite := FALSE;
		END_IF;
		IF tx - last_change >= stage2_delay AND stage2 THEN
			coil2 := TRUE;
		ELSE
			coil2 := FALSE;
		END_IF;
	END_IF;
END_CASE;

(* abschaltung wenn kein eingangssignal *)
IF NOT in THEN
	state := 1;
	motor := FALSE;
	coil1 := FALSE;
	coil2 := FALSE;
	ignite := FALSE;
	pre_heat := FALSE;
	last_change := tx;
END_IF;

(* runtimezähler *)
timer1(in := flame AND in AND motor AND coil1 AND NOT coil2);
timer2(in := flame AND in AND motor AND coil1 AND coil2);
runtime1 := timer1.ontime;
runtime2 := timer2.ontime;
cycles := timer1.cycles;
KWH := runtime1 * KW1 + runtime2 * KW2;

(* zeit fuer naechsten aufruf merken *)
last := tx;

(* set fail output IF ERROR and Status  if normal operation *)

IF status > 0 AND status < 100 THEN
	fail := TRUE;
ELSE
	fail := FALSE;
	IF NOT in THEN
		status := 110;
	ELSIF flame AND in AND motor AND coil2 AND coil1 THEN
		status := 113;
	ELSIF flame AND in AND motor AND coil1 THEN
		status := 112;
	ELSE
		status := 111;
	END_IF;
END_IF;


(*
31.12.2006	hm		rev 1.1
	added pre_heat timing and output
	flame monitor bofe ignition will generate statusure output
	added output for KWh

31.12.2006	hm		rev 1.2
	added oil_temp_input

31.12.2006	hm		rev 1.3
	changed status output to be byte instead of bool

22.1.2007		hm		rev 1.4
	renamed fail output to status
	added output cycles
	renamed 
	corrected an error while pre_heat would be on when an error was present
	added coil2 output and stage2 input
*)
END_FUNCTION_BLOCK

(* POU Byte_of_bit, ST *)
FUNCTION Byte_of_bit : BYTE
VAR_INPUT
	B0:BOOL;
	B1:BOOL;
	B2:BOOL;
	B3:BOOL;
	B4:BOOL;
	B5:BOOL;
	B6:BOOL;
	B7:BOOL;
END_VAR
VAR
	Bx : BYTE;
END_VAR

(*
version 1.0	4 aug 2006
programmer 	hugo
tested by		tobias

this function creates a byte from 8 individual bits

executioin TIME on wago 750-841 = 8 us
*)
BX.0 := B0;
BX.1 := B1;
BX.2 := B2;
BX.3 := B3;
BX.4 := B4;
BX.5 := B5;
BX.6 := B6;
BX.7 := B7;

Byte_of_bit := BX;
END_FUNCTION

(* POU Byte_of_Dword, ST *)
FUNCTION Byte_of_Dword : BYTE
VAR_INPUT
	in : DWORD;
	N : BYTE;
END_VAR
VAR
	temp: DWORD;
END_VAR

(*
version 1.0	17 jan 2007
programmer 	hugo
tested by		tobias

this function extracts a single byte from the nth position from right (right is lowest byte) 
the lower byte (starting with Bit0 from in) is selected with N=0.
*)
temp := SHR(in,n*8);
Byte_of_Dword := DWORD_TO_BYTE(temp);
END_FUNCTION

(* POU Byte_to_Bit, ST *)
FUNCTION_BLOCK Byte_to_Bit
VAR_INPUT
	IN: BYTE;
END_VAR
VAR_OUTPUT
	B0: BOOL;
	B1: BOOL;
	B2: BOOL;
	B3: BOOL;
	B4: BOOL;
	B5: BOOL;
	B6: BOOL;
	B7: BOOL;
END_VAR
VAR
END_VAR

(*
version 1.0	4 aug 2006
programmer 	hugo
tested by		tobias

this Function Block extracts the 8 Bits from a byte

executioin TIME on wago 750-841 = 13us
*)
B0 := IN.0;
B1 := IN.1;
B2 := IN.2;
B3 := IN.3;
B4 := IN.4;
B5 := IN.5;
B6 := IN.6;
B7 := IN.7;
END_FUNCTION_BLOCK

(* POU C_to_F, ST *)
FUNCTION C_to_F : REAL
VAR_INPUT
	celsius : REAL;
END_VAR
VAR
END_VAR

(*
version 1.0	4 aug 2006
programmer 	hugo
tested by		tobias

this function converts celsius  to fahrenheit 

executioin TIME on wago 750-841 = 15us
*)
C_to_F := celsius * 1.8 + 32;
END_FUNCTION

(* POU C_to_K, ST *)
FUNCTION C_to_K : REAL
VAR_INPUT
	Celsius : REAL;
END_VAR
VAR
END_VAR

(*
version 1.0	4 dec 2006
programmer 	hugo
tested by		tobias

this function converts celsius to kelvin
*)
C_to_K := Celsius - 273.15;
END_FUNCTION

(* POU Calibrate, ST *)
FUNCTION_BLOCK Calibrate
VAR_INPUT
	X : REAL;
	CO : BOOL;
	CS : BOOL;
END_VAR
VAR_INPUT CONSTANT
	Y_Offset : REAL;
	Y_Scale : REAL;
END_VAR
VAR_OUTPUT
	Y : REAL;
END_VAR
VAR RETAIN
	offset : REAL;
	Scale : REAL := 1;
END_VAR

(*
	version 1.2	22 feb 2007
	programmer 	hugo
	tested BY		hans

Calibrate allows for offset and scale calibration of an analog input.
offset is calibrated to a stored reference Y_offset while CO is true.
after the offset is calibrated, scale can be calibrated to a reference value Y_scale while CS is true.
*)
(* check for calibration *)
IF CO THEN
	Offset := Y_Offset - X;
ELSIF CS THEN
	scale := Y_scale / (X+Offset);
END_IF;
(* calculate output *)
Y := (X + Offset) * Scale;


(* revision history
hm 22.2.2007		rev 1.2
	changed VAR RETAIN PERSISTENT to VAR RETAIN for better compatibility
	wago lon contollers do not support persisitent

*)
END_FUNCTION_BLOCK

(* POU Offset, ST *)
FUNCTION Offset : REAL
VAR_INPUT
	X : REAL;
	O1, O2, O3, O4 : BOOL;
	D : BOOL;
END_VAR
VAR_INPUT CONSTANT
	Offset_1 : REAL;
	Offset_2 : REAL;
	Offset_3 : REAL;
	Offset_4 : REAL;
	default : REAL;
END_VAR

(*
version 1.0	12 jan 2007
programmer 	oscat
tested by		tobias

The Function offset adds offsets to an analog signal depending on digital inputs.
all selected offsets are added at the same time.
with the input D a default value instead of the input X can be used.

*) 
IF D THEN Offset := default; ELSE Offset := X; END_IF;
IF O1 THEN Offset := Offset + offset_1; END_IF;
IF O2 THEN Offset := Offset + offset_2; END_IF;
IF O3 THEN Offset := Offset + offset_3; END_IF;
IF O4 THEN Offset := Offset + offset_4; END_IF;
END_FUNCTION

(* POU ceil, ST *)
FUNCTION ceil : INT
VAR_INPUT
	X : REAL;
END_VAR
VAR
END_VAR


(*
version 1.0	7 feb 2007
programmer 	hugo
tested by		tobias

This is a rounding function which returns the smallest possible integer which is greater or equal to X.
ceil(3.14) = 4
ceil(-3.14) = 3

*)
ceil := TRUNC(X);
IF ceil < X THEN
	ceil := ceil + 1;
END_IF;
END_FUNCTION

(* POU check_parity, ST *)
FUNCTION check_parity : BOOL
VAR_INPUT
	in : DWORD;
	p : BOOL;
END_VAR
VAR
	i: INT;
	cnt: INT := 0;
END_VAR

(*
version 1.0	1 oct 2006
programmer 	hugo
tested by		tobias

this function checks for an even partity for a dword and partity bit.

*)
FOR i := 0 TO 31 DO
	IF in.0 THEN cnt := cnt +1; END_IF;
	in := SHR(in,1);
END_FOR;
check_parity := even(cnt) XOR P;
END_FUNCTION

(* POU CHR, ST *)
FUNCTION CHR : STRING
VAR_INPUT
	C : BYTE;
END_VAR
VAR
	PT : POINTER TO BYTE;
END_VAR

(*
version 1.0	16 jan 2007
programmer 	hugo
tested by		tobias

CHR creates a character from a byte input and stuffs it in a one character length string.

*)
PT := ADR(CHR);
PT^ := C;
END_FUNCTION

(* POU click, ST *)
FUNCTION_BLOCK click
VAR_INPUT
	in : BOOL;
END_VAR
VAR_OUTPUT
	Q : BOOL;
	single : BOOL;
	double : BOOL;
	triple : BOOL;
	status: BYTE;
END_VAR
VAR_INPUT CONSTANT
	T_debounce : TIME := t#10ms;
	T_short : TIME := t#200ms;
	T_pause : TIME := t#500ms;
	T_reconfig : TIME := t#1m;
END_VAR
VAR
	debounce : TON;
	tx : TIME;
	last : TIME;
	init : BOOL;
	edge : BOOL;
	standby: BOOL;
	state: INT;
END_VAR

(*
version 1.0	15 Feb 2006
programmer 	oscat
tested by		tobias

*)
(* read system time *)
tx := TIME();

(* set last and tx if never started before *)
IF NOT init THEN
	init := TRUE;
	last := tx;
	debounce.PT := T_debounce;
	standby := in;
END_IF;

(* debounce input *)
debounce(in := in XOR standby);
Q := debounce.Q;

(* delete outputs if input is inactive *)
IF NOT Q THEN
	single := FALSE;
	double := FALSE;
	triple := FALSE;
	status := 110;
END_IF;

(* check for input edge *)
IF Q XOR edge THEN
	edge := in;
	last := tx;
	IF Q THEN state := state + 1; END_IF;
END_IF;

IF (q AND tx - last >= T_short) OR (NOT q AND tx - last >= t_pause) THEN
	CASE state OF
		1:	single := TRUE;
			status := 111;
		2:	double := TRUE;
			status := 112;
		3:	triple := TRUE;
			status := 113;
	END_CASE;
	state := 0;
END_IF;

(* determine if high or low active *)
IF tx - last >= t_reconfig AND standby <> in THEN
	standby := in;
END_IF;
END_FUNCTION_BLOCK

(* POU CLK_1ms, ST *)
FUNCTION_BLOCK CLK_1ms
VAR_INPUT
END_VAR
VAR_OUTPUT
	Q : BOOL;
END_VAR
VAR
	CLK : BOOL;
	edge : BOOL := 0;
	stime: DWORD;
END_VAR

(*
clk_gen uses the internal sps time to generate one pulse every 1 ms
every pulse is only valid for one cycle so that a edge trigger is not necessary
clk_gen generates pulses depending on the accuracy of the system clock.

be careful, 1ms clocks will only work on very powerful sps cpu's
wago 750 - 841 will work with pulse width >= 10ms
*)
stime := TIME_TO_DWORD(TIME());
clk := stime.0;
Q := clk XOR edge;
edge := CLK;
END_FUNCTION_BLOCK

(* POU CLK_2ms, ST *)
FUNCTION_BLOCK CLK_2ms
VAR_INPUT
END_VAR
VAR_OUTPUT
	Q : BOOL;
END_VAR
VAR
	CLK : BOOL;
	edge : BOOL := 0;
	stime: DWORD;
END_VAR

(*
clk_gen uses the internal sps time to generate one pulse every 2 ms
every pulse is only valid for one cycle so that a edge trigger is not necessary
clk_gen generates pulses depending on the accuracy of the system clock.

be careful, 1ms clocks will only work on very powerful sps cpu's
wago 750 - 841 will work with pulse width >= 10ms
*)
stime := TIME_TO_DWORD(TIME());
clk := stime.1;
Q := clk XOR edge;
edge := CLK;
END_FUNCTION_BLOCK

(* POU CLK_4ms, ST *)
FUNCTION_BLOCK CLK_4ms
VAR_INPUT
END_VAR
VAR_OUTPUT
	Q : BOOL;
END_VAR
VAR
	CLK : BOOL;
	edge : BOOL := 0;
	stime: DWORD;
END_VAR

(*
clk_gen uses the internal sps time to generate one pulse every 4 ms
every pulse is only valid for one cycle so that a edge trigger is not necessary
clk_gen generates pulses depending on the accuracy of the system clock.

be careful, 1ms clocks will only work on very powerful sps cpu's
wago 750 - 841 will work with pulse width >= 10ms
*)
stime := TIME_TO_DWORD(TIME());
clk := stime.2;
Q := clk XOR edge;
edge := CLK;
END_FUNCTION_BLOCK

(* POU CLK_8ms, ST *)
FUNCTION_BLOCK CLK_8ms
VAR_INPUT
END_VAR
VAR_OUTPUT
	Q : BOOL;
END_VAR
VAR
	CLK : BOOL;
	edge : BOOL := 0;
	stime: DWORD;
END_VAR

(*
clk_gen uses the internal sps time to generate one pulse every 8 ms
every pulse is only valid for one cycle so that a edge trigger is not necessary
clk_gen generates pulses depending on the accuracy of the system clock.

be careful, 1ms clocks will only work on very powerful sps cpu's
wago 750 - 841 will work with pulse width >= 10ms
*)
stime := TIME_TO_DWORD(TIME());
clk := stime.3;
Q := clk XOR edge;
edge := CLK;
END_FUNCTION_BLOCK

(* POU clk_div, ST *)
FUNCTION_BLOCK clk_div
VAR_INPUT
	clk : BOOL;
	rst: BOOL;
END_VAR
VAR_OUTPUT
	Q0 : BOOL := 0;
	Q1 : BOOL := 0;
	Q2 : BOOL := 0;
	Q3 : BOOL := 0;
	Q4 : BOOL := 0;
	Q5 : BOOL := 0;
	Q6 : BOOL := 0;
	Q7 : BOOL := 0;
END_VAR
VAR
	cnt: BYTE := 0;
END_VAR

(*
version 1.0	4 aug 2006
programmer 	hugo
tested by		tobias

this is a clock divider
each output divides the signal by 2
Q0 = clk / 2 , Q1 = Q0 / 2 and so on.
the outputs have a 50% duty cycle each.


*)
IF clk AND NOT rst THEN
	cnt:= cnt +1;
	Q0 := cnt.0;
	Q1 := cnt.1;
	Q2 := cnt.2;
	Q3 := cnt.3;
	Q4 := cnt.4;
	Q5 := cnt.5;
	Q6 := cnt.6;
	Q7 := cnt.7;
END_IF;
IF rst THEN
	cnt:= 0;
	Q0 := 0;
	Q1 := 0;
	Q2 := 0;
	Q3 := 0;
	Q4 := 0;
	Q5 := 0;
	Q6 := 0;
	Q7 := 0;
END_IF;
END_FUNCTION_BLOCK

(* POU CLK_Prg, ST *)
FUNCTION_BLOCK CLK_Prg
VAR_INPUT
	PT : TIME := t#10ms;
END_VAR
VAR_OUTPUT
	Q : BOOL := 0;
END_VAR
VAR
	init : BOOL := FALSE;
	last : TIME;
	tx: TIME;
END_VAR

(*
version 1.1	25 feb 2007
programmer 	hugo
tested by		tobias

clk_prg uses the internal sps time to generate a clock with programmable period time.
the period time is defined for 10ms .. 65s
the first cycle after start is a clk pulse and then depending on the programmed period time a delay.
every pulse is only valid for one cycle.
the accuracy of clk_prg is depending on the accuracy of the system clock.

*)
(* read system time *)
tx := TIME();

(* initialize on startup *)
IF NOT init THEN
	init := TRUE;
	last := tx - pt;
END_IF;

(* generate output pulse when next_pulse is reached *)
IF tx - last >= pt THEN
	Q := TRUE;
	last := tx;
ELSE
	Q := FALSE;
END_IF;


(* revision hiostory

hm 25 feb 2007
	rewritten code for higher performance
	pt can now be changed during runtime
*)
END_FUNCTION_BLOCK

(* POU CLK_Pulse, ST *)
FUNCTION_BLOCK CLK_Pulse
VAR_INPUT
	PT : TIME := t#10ms;
	N : INT := 0;
	rst : BOOL := 0;
END_VAR
VAR_OUTPUT
	Q : BOOL := 0;
	cnt : INT := 0;
	run : BOOL := 0;
END_VAR
VAR
	pti : TIME := t#0ms;
	next_pulse: TIME := T#0s;
	overflow: BOOL := FALSE;
END_VAR

(*
version 1.0	4 aug 2006
programmer 	hugo
tested by		tobias

clk_pulse uses the internal sps time to generate a clock with programmable period time.
the period time is defined for 10ms .. 65s.
pulse generation is continuous if N = 0 and for n pulses otherwise.
if the period time is set to less then 10ms the min clock perid is 10ms.
the first cycle after start is a clk pulse and then depending on the programmed period time a delay.
every pulse is only valid for one cycle so that a edge trigger is not necessary
clk_prg depending on the accuracy of the system clock.

*)
IF rst THEN
	run := FALSE;
	pti := t#0ms;
	next_pulse := t#0ms;
	overflow := FALSE;
	Q := FALSE;
	cnt := 0;
ELSIF cnt <= N OR N = 0 THEN
	IF NOT run THEN
		next_pulse := TIME();
		run := TRUE;
		IF pt < T#10ms THEN PTI := T#10ms; ELSE pti := pt; END_IF;
	END_IF;
	IF TIME() >= next_pulse AND NOT overflow AND (cnt < N OR N = 0) THEN
		Q := TRUE;
		cnt := cnt + 1;
		IF next_pulse + pti < next_pulse THEN
			overflow := TRUE;
		END_IF;
		next_pulse := next_pulse + pti;
	ELSE
		Q := FALSE;
		IF cnt = N THEN run := FALSE; END_IF
		IF TIME() <= next_pulse THEN overflow := FALSE; END_IF;
	END_IF;
END_IF
END_FUNCTION_BLOCK

(* POU cosH, ST *)
FUNCTION cosH : REAL
VAR_INPUT
	X : REAL;
END_VAR
VAR
END_VAR


(*
version 1.0	12 jan 2007
programmer 	hugo
tested by		tobias

this function calculates the cos hyperbolicus

*)
cosH := (EXPT(e,x) + EXPT(e,-x))/2;
END_FUNCTION

(* POU cotH, ST *)
FUNCTION cotH : REAL
VAR_INPUT
	X : REAL;
END_VAR
VAR
END_VAR


(*
version 1.0	12 jan 2007
programmer 	hugo
tested by		tobias

this function calculates the cotangens hyperbolicus

*)
cotH := (EXPT(e, 2 * x) + 1) / (EXPT(e, 2 * x) - 1);
END_FUNCTION

(* POU date_add, ST *)
FUNCTION date_add : DATE
VAR_INPUT
	idate : DATE;
	D : INT;
	W : INT;
	M : INT;
	Y : INT;
END_VAR
VAR
	mo: INT;
	yr : INT;
END_VAR


(*
version 1.0	27 dec 2006
programmer 	hugo
tested by		tobias

date_add adds days, weeks, month or years to a date.
negative inputs are allowed for subtraction.

*)
date_add := DWORD_TO_DATE(DATE_TO_DWORD(idate) + 86400 * d + 604800 * w);
IF y <> 0 THEN
	yr := year(date_add) + y;
END_IF;
IF m > 0 THEN
	mo := month(date_add) + m;
	yr := yr + (mo - 1) / 12;
	mo := mo MOD 12;
	IF mo = 0 THEN mo := 12; END_IF;
	date_add := set_Date(yr, mo, day_of_month(date_add));
ELSIF m < 0 THEN
	mo := month(date_add) + m;
	yr := yr + mo / 12 -1;
	mo := mo MOD 12 + 12;
	date_add := set_Date(yr, mo, day_of_month(date_add));
ELSE
	date_add := set_Date(yr, month(date_add), day_of_month(date_add));
END_IF;
END_FUNCTION

(* POU year, ST *)
FUNCTION year : INT
VAR_INPUT
	idate : DATE;
END_VAR
VAR
END_VAR

(*
version 1.0	4 aug 2006
programmer 	hugo
tested by		tobias

returs the year of a date  
the function works for dates from 1970 - 2099 
execution time on wago 750-841 = 20us   
*)
year := DWORD_TO_INT((DATE_TO_DWORD(idate)/864+71954300)/36525);
END_FUNCTION

(* POU month, ST *)
FUNCTION month : INT
VAR_INPUT
	idate : DATE;
END_VAR
VAR
END_VAR

(*
version 1.0	4 aug 2006
programmer 	hugo
tested by		tobias

returns the month of a date  
execution time on wago 750-841 = 145us
*)
month := STRING_TO_INT(MID(DATE_TO_STRING(idate),2,8));
END_FUNCTION

(* POU set_Date, ST *)
FUNCTION set_Date : DATE
VAR_INPUT
	year : INT;
	month : INT;
	day : INT;
END_VAR
VAR
	count : DWORD;
	leap: BOOL;
END_VAR

(*
version 1.0	4 aug 2006
programmer 	hugo
tested by		tobias

creates a date output from year, month and day of month   
execution time on wago 750-841 = 45 us
*)
IF year MOD 4 = 0 THEN leap := TRUE; ELSE leap := FALSE; END_IF;
count := TRUNC((year-1)*365.25-719178+day);
CASE month OF
2:	count := count + 31;
3:	IF leap THEN count := count + 60; ELSE count := count + 59; END_IF;
4:	IF leap THEN count := count + 91; ELSE count := count + 90; END_IF;
5:	IF leap THEN count := count + 121; ELSE count := count + 120; END_IF;
6:	IF leap THEN count := count + 152; ELSE count := count + 151; END_IF;
7:	IF leap THEN count := count + 182; ELSE count := count + 181; END_IF;
8:	IF leap THEN count := count + 213; ELSE count := count + 212; END_IF;
9:	IF leap THEN count := count + 244; ELSE count := count + 243; END_IF;
10:	IF leap THEN count := count + 274; ELSE count := count + 273; END_IF;
11:	IF leap THEN count := count + 305; ELSE count := count + 304; END_IF;
12:	IF leap THEN count := count + 335; ELSE count := count + 334; END_IF;
END_CASE;
set_Date := DWORD_TO_DATE(count * 86400);
END_FUNCTION

(* POU day_of_month, ST *)
FUNCTION day_of_month : INT
VAR_INPUT
	idate : DATE;
END_VAR
VAR
	yd: INT;
	yr: INT;
END_VAR

(*
version 1.1	22 Jan 2007
programmer 	hugo
tested by		tobias

returns the day OF month from any DATE
execution TIME with wago 750-841 = 65 us
*)
yr := DWORD_TO_INT((DATE_TO_DWORD(idate)/864+71954300)/36525);
yd := DWORD_TO_INT(DATE_TO_DWORD(idate)/86400 - TRUNC((yr-1)*365.25) + 719178);
IF yr MOD 4 = 0 THEN
	CASE yd OF
		1..31 	:	day_of_month := yd;
		32..60	:	day_of_month := yd - 31;
		61..91	:	day_of_month := yd - 60;
		92..121 :	day_of_month := yd - 91;
		122..152:	day_of_month := yd - 121;
		153..182:	day_of_month := yd - 152;
		183..213:	day_of_month := yd - 182;
		214..244:	day_of_month := yd - 213;
		245..274:	day_of_month := yd - 244;
		275..305:	day_of_month := yd - 274;
		306..335:	day_of_month := yd - 305;
		336..366:	day_of_month := yd - 335;
	END_CASE;
	ELSE
	CASE yd OF
		1..31 	:	day_of_month := yd;
		32..59	:	day_of_month := yd - 31;
		60..90	:	day_of_month := yd - 59;
		91..120 :	day_of_month := yd - 90;
		121..151:	day_of_month := yd - 120;
		152..181:	day_of_month := yd - 151;
		182..212:	day_of_month := yd - 181;
		213..243:	day_of_month := yd - 212;
		244..273:	day_of_month := yd - 243;
		274..304:	day_of_month := yd - 273;
		305..334:	day_of_month := yd - 304;
		335..365:	day_of_month := yd - 334;
	END_CASE;
	END_IF;




(*
this function is simple but took too long with 133 us
the problem is date_to_string is far too slow
day_of_month := STRING_TO_INT(RIGHT(DATE_TO_STRING(idate),2));

Revision history

hm 22.1.2007		rev 1.1
	deleted unused variable day_in_year and day_in_year_begin

*)
END_FUNCTION

(* POU day_of_year, ST *)
FUNCTION day_of_year : INT
VAR_INPUT
	idate : DATE;
END_VAR
VAR
END_VAR

(*
version 1.0	4 aug 2006
programmer 	hugo
tested by		tobias

calculates the day of the year 
execution time for wago 750-841 = 44 us  
*)
day_of_year := DWORD_TO_INT(DATE_TO_DWORD(idate)/86400 + 719178 - TRUNC((year(idate)-1)*365.25));
END_FUNCTION

(* POU day_to_time, ST *)
FUNCTION day_to_time : TIME
VAR_INPUT
	input : REAL;
END_VAR
VAR
END_VAR

(*
version 1.0	4 aug 2006
programmer 	hugo
tested by		tobias

converts an amount of days in real to time 
execution time on wago 750-841 =  17 us 
*)
day_to_time := DWORD_TO_TIME(REAL_TO_DWORD(input * 86400000));
END_FUNCTION

(* POU days_delta, ST *)
FUNCTION days_delta : INT
VAR_INPUT
	date_1 : DATE;
	date_2 : DATE;
END_VAR
VAR
END_VAR

(*
version 1.0	27 dec 2006
programmer 	hugo
tested by		tobias

days_delta calculated the days between two dates.

*)
IF date_2 <= date_1 THEN
	days_delta := DWORD_TO_INT((DATE_TO_DWORD(date_1) - DATE_TO_DWORD(date_2)) / 86400);
ELSE
	days_delta := -DWORD_TO_INT((DATE_TO_DWORD(date_2) - DATE_TO_DWORD(date_1)) / 86400);
END_IF;
END_FUNCTION

(* POU DCF77, ST *)
FUNCTION_BLOCK DCF77
VAR_INPUT
	rec : BOOL;
END_VAR
VAR_INPUT CONSTANT
	sync_timeout : TIME := t#2m;
	time_offset : TIME := t#1h;
	dst_en : BOOL := TRUE;
END_VAR
VAR_OUTPUT
	TP : BOOL;
	DST : BOOL;
	weekday : INT;
	error: BOOL := TRUE;
	RTC : DT;
	RTC1 : DT;
	msec : INT;
	sync : BOOL;
END_VAR
VAR
	MEZ : DT;
	UTC : DT;
	state : INT;
	edge: BOOL;
	tx : TIME;
	ty: TIME;
	last : TIME;
	bits : ARRAY[0..58] OF BOOL;
	cnt : INT;
	i : INT;
	old_time : DT;
	minute : INT;
	hour : INT;
	day : INT;
	month : INT;
	year : INT;
	last_sync: TIME;
END_VAR


(*
version 1.2	26 Feb 2007
programmer 	hugo
tested by		tobias

this is a decoder for a DCF77 signal.
the decoder decodes the DCF77 signal and checks for a valid Date_Time.
since the dcf77 signal is only secured with a simple parity the decoder waits for two consecutive valid transmissions before it sets the output signals.
given a valid reception by the receiver the decoder can take up to 3 minutes to start its clocks the first time.
after a valid signal is detected the error output goes low and dignals a valid dcf signal from the receiver.
a tp is only valid for one program cycle to allow for external rtc setting.
after a valid signal is detected two independent internal clocks are started (RTC and RTC1), the seconds  of these clocks are generated by software since the dcf signal is only valid for minutes.
rtc is always utc ( world time) and rtc1 can be set to any time zone by setting the time_zone_offset and enabling dst for automatic summertime.
a sync output signals the the rtc and rtc1 are in sync with the dcf77 signal, if the dcf77 signal is lost for more then the sync time the sync output goes low
but the rtc and rtc1 outputs keep running based on software timing until a valid dcf77 signal is received again and triggers the clock.
in addition a millisecond output gives further resolutionof the clocks.
a dst output shows if daylight saving time is enables and the weekday output shows which day of week currently is ( 1= monday ... 7= sunday).


*)
(* if tp was set it should only be active for 1 cycle *)
TP := FALSE;

IF rec XOR edge THEN
	tx := TIME() - last;
	edge := rec;
	IF NOT rec AND tx > t#1700ms AND tx < t#2000ms THEN
		(* start condition reached *)
		state := 0;
		tp := NOT error;
	ELSIF NOT rec AND tx > t#700ms AND tx < t#1000ms THEN
		(* second switch detected *)
		IF state < 58 THEN state := state +1; ELSE state := 0; END_IF;
	ELSIF rec AND tx  < t#120ms THEN
		(* bit 0 detected  *)
		bits[state] := 0;
	ELSIF rec AND tx > t#120ms AND tx < t#250ms THEN
		(* bit 1 detected *)
		bits[state] := 1;
	ELSE
		(* error condition received signal is not valid *)
		error := TRUE;
		state := 0;
	END_IF;
	last := last + tx;
	IF rec AND state = 58 THEN
		error := FALSE;

		(* decode the bits and check for possible errors *)
		IF bits[0] OR NOT (bits[17] XOR bits[18]) OR NOT bits[20] THEN error := TRUE; END_IF;
		(* decode minute *)
		minute := 0;
		minute.0 := bits[21];
		minute.1 := bits[22];
		minute.2 := bits[23];
		minute.3 := bits[24];
		IF bits[25] THEN minute := minute + 10; END_IF;
		IF bits[26] THEN minute := minute +20; END_IF;
		IF bits[27] THEN minute := minute +40; END_IF;
		IF minute > 59 OR (bits[21] XOR bits[22] XOR bits[23] XOR bits[24] XOR bits[25] XOR bits[26] XOR bits[27] XOR bits[28]) THEN error := TRUE; END_IF;

		(* decode hour *)
		hour := 0;
		hour.0 := bits[29];
		hour.1 := bits[30];
		hour.2 := bits[31];
		hour.3 := bits[32];
		IF bits[33] THEN hour := hour + 10; END_IF;
		IF bits[34] THEN hour := hour +20; END_IF;
		IF hour > 23 OR (bits[29] XOR bits[30] XOR bits[31] XOR bits[32] XOR bits[33] XOR bits[34] XOR bits[35]) THEN error := TRUE; END_IF;

		(* decode day of month *)
		day := 0;
		day.0 := bits[36];
		day.1 := bits[37];
		day.2 := bits[38];
		day.3 := bits[39];
		IF bits[40] THEN day := day + 10; END_IF;
		IF bits[41] THEN day := day + 20; END_IF;
		IF day > 31 THEN error := TRUE; END_IF;

		(* decode day of week *)
		weekday := 0;
		weekday.0 := bits[42];
		weekday.1 := bits[43];
		weekday.2 := bits[44];
		IF weekday > 7 OR weekday < 1 THEN error := TRUE; END_IF;

		(* decode month *)
		month := 0;
		month.0 := bits[45];
		month.1 := bits[46];
		month.2 := bits[47];
		month.3 := bits[48];
		IF bits[49] THEN month := month +10; END_IF;
		IF month > 12 THEN error := TRUE; END_IF;

		(* decode year *)
		year := 0;
		year.0 := bits[50];
		year.1 := bits[51];
		year.2 := bits[52];
		year.3 := bits[53];
		IF bits[54] THEN year := year + 10; END_IF;
		IF bits[55] THEN year := year + 20; END_IF;
		IF bits[56] THEN year := year + 40; END_IF;
		IF bits[57] THEN year := year + 80; END_IF;

		(* check parity for bits 36 to 58 *)
		cnt := 0;
		FOR i := 36 TO 58 DO IF bits[i] THEN cnt := cnt + 1; END_IF; END_FOR;
		IF NOT even(cnt) THEN error := TRUE; END_IF;

		(* time must be valid for two cycles to clear error flag *)
		IF NOT error THEN
			(* set outputs *)
			old_time := mez;
			IF year >= 70 THEN year := year + 1900; ELSE year := year + 2000; END_IF;
			mez := set_DT(year,month,day,hour,minute,0);
			DST := bits[17];
			IF DST THEN
				UTC := DWORD_TO_DT(DT_TO_DWORD(mez) - 7200);
			ELSE
				UTC := DWORD_TO_DT(DT_TO_DWORD(mez) - 3600);
			END_IF

			(* set trigger signal only if the receiver has received 2 successive minutes *)
			IF mez <> old_time + t#1m THEN error := TRUE ; END_IF;
		END_IF;
	END_IF;
END_IF;

(* this portion implements a free running clock which is triggered by the dcf77 signal *)
IF tp THEN
	rtc := utc;
	IF DST AND dst_en THEN rtc1 := rtc + time_offset + t#1h; ELSE rtc1 := rtc + time_offset; END_IF;
	sync := TRUE;
	last_sync := last;
	ty := last;
ELSIF rtc > DWORD_TO_DT(0) AND TIME() - ty >= t#1s THEN
	rtc := rtc + t#1s;
	rtc1 := rtc1 + t#1s;
	ty := ty + t#1s;
	sync := ty - last_sync < sync_timeout AND last_sync > DWORD_TO_TIME(0);
	weekday := weekday(DT_TO_DATE(rtc1));
	DST := dst_en AND DST(utc, time_offset);
END_IF;
msec := TIME_TO_INT(TIME() - ty);



(* decode information
bits		content
0			Bitwert immer 0
1 bis 14	reserviert für Betriebsinformationen (nicht für DCF77-Nutzer bestimmt)
15			Rufbit für Alarmierung der PTB-Mitarbeiter
			(bis Mai 2003: Bitwert = 0 falls normale Antenne in Verwendung; 1 = Backupantenne)
16			Bitwert = 1 falls ein Wechsel von MEZ nach MESZ oder umgekehrt bevorsteht; Dauer der Anzeige: 1 Stunde
17 + 18	gültige Zeit = MEZ, falls Bit 17=0 und Bit 18=1
			gültige Zeit = MESZ, falls Bit 17=1 und Bit 18=0
19			Bitwert = 1 falls innerhalb den nächsten 59 Minuten eine Schaltsekunde angeordnet ist. Beim Einfügen einer Schaltsekunde wird anstelle der 59. die 60. Sekundenmarke weggelassen und in der 58. erfolgt ausnahmsweise ein Trägerabfall.
20			Startbit für Zeitinformation (immer 1)
21 - 27		1, 2, 4, 8, 10, 20, 40 Minuten (bitweise Addition)
28			Prüfbit (gerade Parität) für die Bits 21-27
29 - 34		1, 2, 4, 8, 10, 20 Stunden (bitweise Addition)
35			Prüfbit (gerade Parität) für die Bits 29-34
36 - 41		Tagesnummer im aktuellen Monat: 1, 2, 4, 8, 10, 20 (bitweise Addition)
42 - 44		Tagesnummer in der aktuellen Woche: 1, 2, 4 (bitweise Addition)
45 - 49		Monatsnummer: 1, 2, 4, 8, 10 (bitweise Addition)
50 - 57		Jahr (zweistellig): 1, 2, 4, 8, 10, 20, 40, 80 (bitweise Addition)
58			Prüfbit (gerade Parität) füR die Bits 36-57

*)
(* revision history

hm 2.feb 2007		rev 1.1
	change wday and dst outputs when there is no dcf reception

hm	26.feb 2007	rev 1.2
	changed statements where t#1h would be substracted from DT.
	under certain conditions the compiler would crash translating this statement
*)
END_FUNCTION_BLOCK

(* POU DST, ST *)
FUNCTION DST : BOOL
VAR_INPUT
	utc : DT;
	time_zone_offset : TIME;
END_VAR
VAR
	yr : INT;
	yr4 : DWORD;
	ltc: DWORD;
	idate : DWORD;
END_VAR

(*
version 1.0	4 aug 2006
programmer 	hugo
tested by		tobias

 this functions returns TRUE IF dst TIME is active 
 the FUNCTION calculates automaticall FOR any year betweek 1970 AND 2099 
wheather daylight savings is on OR off 
the summertime calculation is done according to european standards.
dst will become TRUE AT 02:00 in the morning FOR the respective days 
AND it will become FALSE after daylight savings TIME is switched back end OF october automatically 
(execution TIME on wago 750-841 =  110us   
*)
yr := year(DT_TO_DATE(utc));
ltc := DT_TO_DWORD(utc+time_zone_offset);
idate := DT_TO_DWORD(set_DT(yr,3,31,2,0,0));
yr4 := 5*yr/4;
IF idate - ((yr4+4) MOD 7)*86400 <= ltc AND idate + (214 - (yr4+1) MOD 7)*86400 > ltc THEN DST := TRUE; ELSE DST := FALSE; END_IF;


(*

Equation used TO calculate the beginning OF European Summer TIME:
Sunday (31 - (5*y/4 + 4) mod 7) March at 01.00 UTC
(valid through 2099, courtesy of Robert H. van Gent, EC).

European Summer Time ends (clocks go back) at 01.00 UTC on

    * 29 October 2006
    * 28 October 2007
    * 26 October 2008

Equation used to calculate the end of European Summer Time:
Sunday (31 - (5*y/4 + 1) mod 7) October at 01.00 UTC
(validity AND credits as above).

*)
END_FUNCTION

(* POU set_DT, ST *)
FUNCTION set_DT : DT
VAR_INPUT
	year : INT;
	month : INT;
	day : INT;
	hour : INT;
	minute : INT;
	second : INT;
END_VAR
VAR
	count : DWORD;
	leap : BOOL;
END_VAR

(*
version 1.0	4 aug 2006
programmer 	hugo
tested by		tobias


creates a date output from year, month and day of month
year must be in the form of 4 digits ie 2006 or 1977.
execution time on wago 750-841 = 45 us   
*)
IF year MOD 4 = 0 THEN leap := TRUE; ELSE leap := FALSE; END_IF;
count := TRUNC((year-1)*365.25-719178+day);
CASE month OF
2:	count := count + 31;
3:	IF leap THEN count := count + 60; ELSE count := count + 59; END_IF;
4:	IF leap THEN count := count + 91; ELSE count := count + 90; END_IF;
5:	IF leap THEN count := count + 121; ELSE count := count + 120; END_IF;
6:	IF leap THEN count := count + 152; ELSE count := count + 151; END_IF;
7:	IF leap THEN count := count + 182; ELSE count := count + 181; END_IF;
8:	IF leap THEN count := count + 213; ELSE count := count + 212; END_IF;
9:	IF leap THEN count := count + 244; ELSE count := count + 243; END_IF;
10:	IF leap THEN count := count + 274; ELSE count := count + 273; END_IF;
11:	IF leap THEN count := count + 305; ELSE count := count + 304; END_IF;
12:	IF leap THEN count := count + 335; ELSE count := count + 334; END_IF;
END_CASE;
set_DT := DWORD_TO_DT(count * 86400 + second + minute * 60 + hour * 3600);
END_FUNCTION

(* POU hour, ST *)
FUNCTION hour : INT
VAR_INPUT
	itod : TOD;
END_VAR
VAR
END_VAR

(*
version 1.0	4 aug 2006
programmer 	hugo
tested by		tobias

extracts the hour of a Time_of_day 
execution time for wago 750-841 = 10 us  
*)
hour := DWORD_TO_INT(TOD_TO_DWORD(itod)/3600000);




(* change history

2.10.2006 changes name of input to itod

*)
END_FUNCTION

(* POU minute, ST *)
FUNCTION minute : INT
VAR_INPUT
	itod : TOD;
END_VAR
VAR
END_VAR

(*
version 1.1	2 oct 2006
programmer 	hugo
tested by		tobias

extracts the minutes out of TOD truncating the ceconds 
execution time on wago 750-841  = 18us

*)  
minute := DWORD_TO_INT(TOD_TO_DWORD(itod)/60000 - TOD_TO_DWORD(itod)/3600000 * 60);


(* change history

2.10.2006 changes name of input to itod

*)
END_FUNCTION

(* POU second, ST *)
FUNCTION second : REAL
VAR_INPUT
	itod : TOD;
END_VAR
VAR
END_VAR

(*
version 1.1	2 oct 2006
programmer 	hugo
tested by		tobias

returns the seconds and milliseconds as real of TOD   
execution time on wago 750-841 = 20 us 
*)
second := DWORD_TO_REAL(TOD_TO_DWORD(itod) - TOD_TO_DWORD(itod)/60000 * 60000)/1000;



(* change history

2.10.2006 changes name of input to itod

*)
END_FUNCTION

(* POU weekday, ST *)
FUNCTION weekday : INT
VAR_INPUT
	idate : DATE;
END_VAR
VAR
END_VAR

(*
version 1.1	21 aug 2006
programmer 	hugo
tested by		tobias

calculates the weekday of a week   
monday = 1 ..... sunday = 7  
execution time on wago 750-841 = 22 us  
*)
weekday := DWORD_TO_INT((DATE_TO_DWORD(idate)/86400+3) MOD 7)+1;

(* corrected a miscalculation formula is now correct *)
END_FUNCTION

(* POU dead_zone, ST *)
FUNCTION dead_zone : REAL
VAR_INPUT
	X : REAL;
	L : REAL;
END_VAR
VAR
END_VAR

(*
version 1.0	12 Feb 2007
programmer 	hugo
tested by		tobias

dead_zone2 is a linear transfer function which follows a linear function except for x is close to 0.
Y = X if abs(x) > L otherwise its 0.

*)
IF ABS(x) > L THEN
	dead_zone := X;
ELSE
	dead_zone := 0;
END_IF;
END_FUNCTION

(* POU dead_zone2, ST *)
FUNCTION_BLOCK dead_zone2
VAR_INPUT
	X : REAL;
	L : REAL;
END_VAR
VAR_OUTPUT
	Y: REAL;
END_VAR
VAR
END_VAR

(*
version 1.0	12 Feb 2007
programmer 	hugo
tested by		tobias

dead_zone2 is a linear transfer function which follows a linear function except for x is close to 0.
Y = X if abs(x) > L.
for values of 0 +/. L a hysteresis function will hold the output at + or - L.

*)
IF ABS(x) > L THEN
	Y := X;
ELSIF Y > 0 THEN
	Y := L;
ELSE
	Y := -L;
END_IF;
END_FUNCTION_BLOCK

(* POU DEC_2, ST *)
FUNCTION_BLOCK DEC_2
VAR_INPUT
	D: BOOL;
	A: BOOL;
END_VAR
VAR_OUTPUT
	Q0: BOOL;
	Q1: BOOL;
END_VAR
VAR
END_VAR

(*
version 1.1	3 Mar 2007
programmer 	hugo
tested by		tobias

a bit input will be decoded to the two outputs Q0 or Q1
dependent on the value of A
A=0 decodes to Q0 and A=1 decodes to Q1

*)
Q0 := D AND NOT A;
Q1 := D AND A;

(* revision history
hm 3.3.2007	rev 1.0
	rewritten in ST for better compatibility

*)
END_FUNCTION_BLOCK

(* POU DEC_4, ST *)
FUNCTION_BLOCK DEC_4
VAR_INPUT
	D: BOOL;
	A0: BOOL;
	A1: BOOL;
END_VAR
VAR_OUTPUT
	Q0: BOOL;
	Q1: BOOL;
	Q2: BOOL;
	Q3: BOOL;
END_VAR
VAR
END_VAR

(*
version 1.1	3 Mar 2007
programmer 	hugo
tested by		tobias

a bit input will be decoded to one of the 4 outputs
dependent on the Adress on A0 and A1

executioin TIME on wago 750-841 = 9us
*)
Q0 := D AND NOT A0 AND NOT A1;
Q1 := D AND A0 AND NOT A1;
Q2 := D AND NOT A0 AND A1;
Q3 := D AND A0 AND A1;

(* revision history
hm 3.3.2007	rev 1.0
	rewritten in ST for better compatibility

*)
END_FUNCTION_BLOCK

(* POU DEC_8, ST *)
FUNCTION_BLOCK DEC_8
VAR_INPUT
	D: BOOL;
	A0: BOOL;
	A1: BOOL;
	A2: BOOL;
END_VAR
VAR_OUTPUT
	Q0: BOOL;
	Q1: BOOL;
	Q2: BOOL;
	Q3: BOOL;
	Q4: BOOL;
	Q5: BOOL;
	Q6: BOOL;
	Q7: BOOL;
END_VAR
VAR
END_VAR

(*
version 1.1	3 mar 2007
programmer 	hugo
tested by		tobias

a bit input will be decoded to one of the 8 outputs
dependent on the Adress on A0, A1 and A2

executioin TIME on wago 750-841 = 17us
*)
Q0 := D AND NOT A0 AND NOT A1 AND NOT A2;
Q1 := D AND A0 AND NOT A1 AND NOT A2;
Q2 := D AND NOT A0 AND A1 AND NOT A2;
Q3 := D AND A0 AND A1 AND NOT A2;
Q4 := D AND NOT A0 AND NOT A1 AND A2;
Q5 := D AND A0 AND NOT A1 AND A2;
Q6 := D AND NOT A0 AND A1 AND A2;
Q7 := D AND A0 AND A1 AND A2;

(* revision history
hm 3.3.2007	rev 1.0
	rewritten in ST for better compatibility

*)
END_FUNCTION_BLOCK

(* POU deg, ST *)
FUNCTION deg : REAL
VAR_INPUT
	rad : REAL;
END_VAR
VAR
END_VAR
VAR
END_VAR

(*
version 1.0	4 aug 2006
programmer 	hugo
tested by		tobias

this function converts degrees into Radiant
execution time on wago 750 - 841 =  10  us
*)
deg := 57.29577951308232 * Rad;
END_FUNCTION

(* POU Rad, ST *)
FUNCTION Rad : REAL
VAR_INPUT
	deg : REAL;
END_VAR
VAR
END_VAR

(*
version 1.0	4 aug 2006
programmer 	hugo
tested by		tobias

this function converts Radiant to degrees
execution time on wago 750 - 841 =  10  us
*)
Rad := 0.0174532925199433 * deg;
END_FUNCTION

(* POU delay, ST *)
FUNCTION_BLOCK delay
VAR_INPUT
	in : REAL;
	N : INT;
	rst : BOOL;
END_VAR
VAR_OUTPUT
	out : REAL;
END_VAR
VAR
	buf : ARRAY[0..31] OF REAL;
	i : INT;
END_VAR

(*
version 1.2	19. jan 2007
programmer 	hugo
tested by		tobias

this function block delays input values by each programm cycle
after N+1 cycles the in value has shifted to the out.
N can be any alue from 0 .. 32
if n = 0 the input will be present on the output without a delay.
f N > 32 then the output will be delayed by 32 cycles.
any high on rst will load the buffer with in.

*)
IF N > SIZEOF(buf) / SIZEOF(in) THEN N:= 32; END_IF;
IF rst THEN
	FOR i := 0 TO 31 DO buf[i] := 0; END_FOR;
	out := in;
ELSIF N < 1 THEN out := in;
ELSE
	IF i >= N THEN i := 0; END_IF;
	out := buf[i];
	buf[i] := in;
	i := i + 1;
END_IF;

(* revision history
hm 1.10.2006	rev 1.1
	corrected error in buffer management

hm 19.1.2007	rev 1.2
	changed reset to load in instead of 0

*)
END_FUNCTION_BLOCK

(* POU delay_4, ST *)
FUNCTION_BLOCK delay_4
VAR_INPUT
	in : REAL;
END_VAR
VAR_OUTPUT
	out1 : REAL;
	out2 : REAL;
	out3 : REAL;
	out4 : REAL;
END_VAR
VAR
	temp: REAL;
END_VAR

(*
version 1.1	19 jan 2007
programmer 	hugo
tested by		tobias

this function block delays input values by each programm cycle
after 4 cycles the in value has shifted to the out 4 and will be discarded after the next cycle
the blocks can be cascaded.

*)
out4 := out3;
out3 := out2;
out2 := out1;
out1 := temp;
temp := in;

(* revision history

hm 19.1.2007	rev 1.1
	added variable temp to add 1 delay  for q1

*)
END_FUNCTION_BLOCK

(* POU dew_temp, ST *)
FUNCTION dew_temp : REAL
VAR_INPUT
	RH : REAL;
	T : REAL;
END_VAR
VAR
	a : REAL := 7.5;
	b : REAL := 237.3;
	SDD : REAL;
	DD : REAL;
	V : REAL;
END_VAR

(*
version 1.0	2 oct 2006
programmer 	hugo
tested by		tobias

this function calculates the deew point for air given the temperature and relative humidity.
dew_temp(60,25) = 16.7 °C.
which means the dew point for air with 25° and 60% RH is at 16.7 °C.


*)
SDD := 6.1078*EXPT(10,(a*T)/(b+T));
DD := RH/100 * SDD;
V := LOG(DD/6.1078);
dew_temp := b*V/(a-v);

(*
Bezeichnungen:
r = relative Luftfeuchte
T = Temperatur in °C
TK = Temperatur in Kelvin (TK = T + 273.15)
TD = Taupunkttemperatur in °C
DD = Dampfdruck in hPa
SDD = Sättigungsdampfdruck in hPa

Parameter:
a = 7.5, b = 237.3 für T >= 0
a = 7.6, b = 240.7 für T < 0 über Wasser (Taupunkt)
a = 9.5, b = 265.5 für T < 0 über Eis (Frostpunkt)

R* = 8314.3 J/(kmol*K) (universelle Gaskonstante)
mw = 18.016 kg (Molekulargewicht des Wasserdampfes)
AF = absolute Feuchte in g Wasserdampf pro m3 Luft

Formeln:

   1. SDD(T) = 6.1078 * 10^((a*T)/(b+T))
   2. DD(r,T) = r/100 * SDD(T)
   3. r(T,TD) = 100 * SDD(TD) / SDD(T)
   4. TD(r,T) = b*v/(a-v) mit v(r,T) = log10(DD(r,T)/6.1078)
   5. AF(r,TK) = 10^5 * mw/R* * DD(r,T)/TK; AF(TD,TK) = 10^5 * mw/R* * SDD(TD)/TK 

*)
END_FUNCTION

(* POU dimm_i, ST *)
FUNCTION_BLOCK dimm_i
VAR_INPUT
	set : BOOL;
	in : BOOL;
	rst : BOOL;
END_VAR
VAR_INPUT CONSTANT
	T_debounce : TIME := T#10ms;
	T_reconfig : TIME := T#10s;
	T_on_max : TIME := T#0h;
	T_dimm_start : TIME := T#1s;
	T_dimm: TIME := T#3s;
END_VAR
VAR_OUTPUT
	Q : BOOL := 0;
	out : BYTE := 0;
END_VAR
VAR
	tx : TIME := T#0s;
	last_edge : BOOL;
	state : BYTE := 0;
	edge : BOOL := 0;
	r_edge : BOOL := 0;
	T_on : TIME;
	dimm_up: BOOL;
	last_step : TIME;
	tn: TIME;
END_VAR

(*
version 1.2	2 Feb 2007
programmer 	hugo
tested by		tobias

this is an intelligent dimmer interface with an autoset feature for "in" it will automatically detect the type of switch:
low active pulses or high high active pulses are allowd for in.
a configurable debounce timer will debounce input signals
if t_on_max is set to anything other then 0 the output will be turned off after the max on time is reached.
the times for debounce, dimming ramp, wait time before dimming and max on time are all programmable.

the dimmer has outputs Q for on and off and also out with the analog dimm value.

*)
(* read system time *)
tn := TIME();

IF rst THEN
	state := 0;
	Q := 0;
	dimm_up := TRUE;
ELSIF set THEN
	state := 0;
	Q := TRUE;
	out := 255;
	dimm_up := FALSE;
	T_on := Tn;
ELSE
	CASE state OF
	(* state 0 wait for activity *)
	0 :	IF (r_edge AND in AND NOT edge) OR (NOT r_edge AND NOT in AND edge) THEN
			IF t_debounce = t#0s THEN state := 2;  ELSE state := 1; END_IF;
			tx := Tn;
			last_edge := in;
		END_IF

	(* state 1 debouncing *)
	1:	IF Tn - T_debounce >= tx THEN
			state := 2;
			tx := Tn;
		END_IF;

	(* state 2 wait for second edge to toggle output *)
	2:	IF Tn - T_dimm_start >= tx THEN
			state := 3;
			tx := Tn;
			(* time to switch elapsed without switching if Q = 0 turn on output and start dimming at 1 *)
			IF NOT Q THEN
				Q := TRUE;
				t_on := tx;
				out := 1;
				dimm_up := TRUE;
			ELSE
				IF out =255 THEN dimm_up := FALSE; END_IF;
			END_IF;
		ELSIF in XOR edge THEN
			(* wait for edge to toggle output and stop all activity *)
			IF Q THEN
				Q := FALSE;
				state := 0;
			ELSE
				Q := TRUE;
				state := 3;
				IF out = 0 THEN out := 255; END_IF
				IF out = 255 THEN dimm_up := FALSE; END_IF;
				tx := Tn;
				t_on := tx;
			END_IF;
		END_IF;

	(* state 3 entered dimming phase *)
	3:	IF in AND r_edge THEN
			(* generate ramp *)
			tx := Tn;
			IF tx >= last_step + T_dimm / 255 THEN
				last_step := tx;
				IF dimm_up AND out < 255 THEN
					out := out + 1;
					IF out = 255 THEN
						dimm_up := FALSE;
						state := 0;
					END_IF;
				ELSIF NOT dimm_up AND out > 0 THEN
					out := out -1;
					IF out = 0 THEN
						Q := FALSE;
						state := 0;
						dimm_up := TRUE;
					 END_IF;
				 END_IF;
			END_IF;
		ELSE
			dimm_up := NOT dimm_up;
			state := 0;
		END_IF;

	END_CASE;

	(* check for max t_on time and reset output if too long *)
	IF Q AND t_on_max > T#0s AND Tn - t_on_max >= T_on THEN Q := 0; END_IF;

	(* check for reconfig and set R_edge to high for rising edge sensitivity *)
	IF Tn - T_reconfig >= tx THEN R_edge := NOT in; END_IF;

	(* set edge to follow in for next edge detection *)
	edge := in;
END_IF;


(* revision history

hm 22.1.2007		rev 1.1
	deleted unused structure ramp

hm 2.feb 2007		rev 1.2
	changed structure to read time() at the beginning for better time consistency if a higher priorized tak interrupts dimm_i
	added statements in case structure for state 1 to allow for short 1 cycle input pulses
*)
END_FUNCTION_BLOCK

(* POU DWord_of_Byte, ST *)
FUNCTION DWord_of_Byte : DWORD
VAR_INPUT
	B0 : BYTE;
	B1 : BYTE;
	B2 : BYTE;
	B3 : BYTE;
END_VAR
VAR
END_VAR

(*
version 1.0	24 jan 2007
programmer 	hugo
tested by		tobias

this function creates a Dword from 4 individual bytes

*)
DWord_of_Byte := B3;
DWord_of_Byte := SHL(DWord_of_Byte,8) + B2;
DWord_of_Byte := SHL(DWord_of_Byte,8) + B1;
DWord_of_Byte := SHL(DWord_of_Byte,8) + B0;
END_FUNCTION

(* POU DWORD_To_STRF, ST *)
FUNCTION DWORD_To_STRF : STRING
VAR_INPUT
	IN : DWORD;
	N : INT;
END_VAR
VAR
	L: INT;
	temp: STRING;
END_VAR

(*
version 1.0	26 jan 2007
programmer 	hugo
tested by		tobias

dword_to_strF converts a DWORD, BYTE or Word to a fixed length String.
the string will be filles with leading zeroes to achieve the fixed length, or if too long, the lowest digits will be used.

for example:	dword_to_strf(123,4) = '0123' 
				dword_to_strf(123,2) = '23'
*)
(* convert dword to string first and cut to length N *)
temp := RIGHT(DWORD_TO_STRING(in),N);
L := LEN(temp);
WHILE L < N DO
	temp := CONCAT('0', temp);
	L := L + 1;
END_WHILE;
DWORD_To_STRF := temp;
END_FUNCTION

(* POU easter, ST *)
FUNCTION easter : DATE
VAR_INPUT
	year : INT;
END_VAR
VAR
	A: INT;
	B: INT;
	C: INT;
	D: INT;
	e: INT;
	f: INT;
	g: INT;
	h: INT;
	i: INT;
	k: INT;
	l: INT;
	m: INT;
	n: INT;
	o: INT;
END_VAR

(*
version 1.0	27 dec 2006
programmer 	hugo
tested by		tobias

easter calculates the day of easter sunday for a given year.
most other catholic holidays are calculated in reference to easter sunday.

*)
a := year MOD 19;
b := year / 100;
c := year MOD 100;
d := b / 4;
e := b MOD 4;
f :=	(b + 8) / 25;
g := (b - f + 1) / 3;
h := (19 * a + b - d - g + 15) MOD 30;
i :=	c / 4;
k := c MOD 4;
l := (32 + 2 * e + 2 * i - h - k) MOD 7;
m := (a + 11 * h + 22 * l) / 451;
n := (h + l - 7 * m + 114) / 31;
o := (h + l - 7 * m + 114) MOD 31;

easter := set_Date(year,n,o+1);

(*
Im Magazin "Nature" vom 20. April 1876 veröffentlichte ein anonymer Autor eine Tabelle mit Regeln zur Berechnung des (Gregorianischen) Ostersonntages des Jahres J. In Formeln ausgedrückt erhält man das Folgende:
a	=	J mod 19
b	=	int(J / 100)
c	=	J mod 100
d	=	int(b / 4)
e	=	b mod 4
f	=	int((b + 8) / 25)
g	=	int((b - f + 1) / 3
h	=	(19 · a + b - d - g + 15) mod 30
i	=	int(c / 4)
k	=	c mod 4
l	=	(32 + 2 · e + 2 · i - h - k) mod 7
m	=	int((a + 11 · h + 22 · l) / 451)
n	=	int((h + l - 7 · m + 114) / 31)
o	=	(h + l - 7 · m + 114) mod 31

n ist hierbei die Nummer des Monats, o + 1 die Nummer des Tages auf welchen der Ostersonntag im Jahr J fällt. Dieser Algorithmus kommt ohne Hilfszahlen aus.

*)
END_FUNCTION

(* POU ESR_collect, ST *)
FUNCTION_BLOCK ESR_collect
VAR_INPUT
	ESR_0, ESR_1, ESR_2, ESR_3, ESR_4, ESR_5, ESR_6, ESR_7 : ARRAY [0..3] OF esr_data;
END_VAR
VAR_OUTPUT
	ESR_OUT : ARRAY[0..63] OF esr_data;
	pos : INT;
END_VAR
VAR CONSTANT
	max_in : INT := 3; (* maximum element of input variable *)
	max_out : INT := 63; (* maximum element of output array *)
END_VAR
VAR
	cnt : INT;
END_VAR

(*
version 1.0	26 jan 2007
programmer 	hugo
tested by		tobias

ESR_collect collects esr data from up to 8 esr_mon modules and stroes them in an output array.
the output pos will display the position of the last element in the array.
if the array will be full, the oldest element is overwritten.

*)
FOR cnt := 0 TO max_in DO
	IF esr_0[cnt].typ > 0 THEN
		esr_out[pos] := esr_0[cnt];
		pos := pos + 1;
		IF pos > max_out THEN pos := 0; END_IF;
	END_IF;
END_FOR;
FOR cnt := 0 TO max_in DO
	IF esr_1[cnt].typ > 0 THEN
		esr_out[pos] := esr_1[cnt];
		pos := pos + 1;
		IF pos > max_out THEN pos := 0; END_IF;
	END_IF;
END_FOR;
FOR cnt := 0 TO max_in DO
	IF esr_2[cnt].typ > 0 THEN
		esr_out[pos] := esr_2[cnt];
		pos := pos + 1;
		IF pos > max_out THEN pos := 0; END_IF;
	END_IF;
END_FOR;
FOR cnt := 0 TO max_in DO
	IF esr_3[cnt].typ > 0 THEN
		esr_out[pos] := esr_3[cnt];
		pos := pos + 1;
		IF pos > max_out THEN pos := 0; END_IF;
	END_IF;
END_FOR;
FOR cnt := 0 TO max_in DO
	IF esr_4[cnt].typ > 0 THEN
		esr_out[pos] := esr_4[cnt];
		pos := pos + 1;
		IF pos > max_out THEN pos := 0; END_IF;
	END_IF;
END_FOR;
FOR cnt := 0 TO max_in DO
	IF esr_5[cnt].typ > 0 THEN
		esr_out[pos] := esr_5[cnt];
		pos := pos + 1;
		IF pos > max_out THEN pos := 0; END_IF;
	END_IF;
END_FOR;
FOR cnt := 0 TO max_in DO
	IF esr_6[cnt].typ > 0 THEN
		esr_out[pos] := esr_6[cnt];
		pos := pos + 1;
		IF pos > max_out THEN pos := 0; END_IF;
	END_IF;
END_FOR;
FOR cnt := 0 TO max_in DO
	IF esr_7[cnt].typ > 0 THEN
		esr_out[pos] := esr_7[cnt];
		pos := pos + 1;
		IF pos > max_out THEN pos := 0; END_IF;
	END_IF;
END_FOR;
END_FUNCTION_BLOCK

(* POU ESR_MON_B8, ST *)
FUNCTION_BLOCK ESR_MON_B8
VAR_INPUT
	s0, s1, s2, s3, s4, s5, s6, s7 : BOOL;
	DT_in : DT;
END_VAR
VAR_INPUT CONSTANT
	a0, a1, a2, a3, a4, a5, a6, a7 : STRING(10);
END_VAR
VAR_OUTPUT
	ESR_Out: ARRAY [0..3] OF esr_data;
	ESR_Flag : BOOL;
END_VAR
VAR
	x0, x1, x2, x3, x4, x5, x6, x7 : BOOL;
	tx: TIME;
	cnt : INT;
END_VAR

(*
version 1.0	26 jan 2007
programmer 	hugo
tested by		tobias

ESR_mon_B8 monitores up to 8 binary inputs and reports changes with time stamd and adress label.
the module checks 8 inputs for a change and reports all changes with time and adress stamp to the output.
4 events maximum can be collected at once within the same cycle

*)
(* read system timer *)
tx := TIME();
ESR_Flag := FALSE;
esr_out[3].typ := 0;
esr_out[2].typ := 0;
esr_out[1].typ := 0;
esr_out[0].typ := 0;
cnt := 0;

(* check if inputs have chaged and fill buffer *)
IF s0 <> X0 THEN
	IF s0 THEN esr_out[cnt].typ := 11; ELSE 	esr_out[cnt].typ := 10; END_IF;
	esr_out[cnt].adress := a0;
	esr_out[cnt].DS := DT_in;
	esr_out[cnt].TS := TX;
	X0 := S0;
	cnt := cnt + 1;
	esr_flag := TRUE;
END_IF;
IF s1 <> X1 THEN
	IF s1 THEN esr_out[cnt].typ := 11; ELSE 	esr_out[cnt].typ := 10; END_IF;
	esr_out[cnt].adress := a1;
	esr_out[cnt].DS := DT_in;
	esr_out[cnt].TS := TX;
	X1 := S1;
	cnt := cnt + 1;
	esr_flag := TRUE;
END_IF;
IF s2 <> X2 THEN
	IF s2 THEN esr_out[cnt].typ := 11; ELSE 	esr_out[cnt].typ := 10; END_IF;
	esr_out[cnt].adress := a2;
	esr_out[cnt].DS := DT_in;
	esr_out[cnt].TS := TX;
	X2 := S2;
	cnt := cnt + 1;
	esr_flag := TRUE;
END_IF;
IF s3 <> X3 THEN
	IF s3 THEN esr_out[cnt].typ := 11; ELSE 	esr_out[cnt].typ := 10; END_IF;
	esr_out[cnt].adress := a3;
	esr_out[cnt].DS := DT_in;
	esr_out[cnt].TS := TX;
	X3 := S3;
	cnt := cnt + 1;
	esr_flag := TRUE;
END_IF;
IF s4 <> X4 AND cnt < 4 THEN
	IF s4 THEN esr_out[cnt].typ := 11; ELSE 	esr_out[cnt].typ := 10; END_IF;
	esr_out[cnt].adress := a4;
	esr_out[cnt].DS := DT_in;
	esr_out[cnt].TS := TX;
	X4 := S4;
	cnt := cnt + 1;
	esr_flag := TRUE;
END_IF;
IF s5 <> X5  AND cnt < 4 THEN
	IF s5 THEN esr_out[cnt].typ := 11; ELSE 	esr_out[cnt].typ := 10; END_IF;
	esr_out[cnt].adress := a5;
	esr_out[cnt].DS := DT_in;
	esr_out[cnt].TS := TX;
	X5 := S5;
	cnt := cnt + 1;
	esr_flag := TRUE;
END_IF;
IF s6 <> X6  AND cnt < 4 THEN
	IF s6 THEN esr_out[cnt].typ := 11; ELSE 	esr_out[cnt].typ := 10; END_IF;
	esr_out[cnt].adress := a6;
	esr_out[cnt].DS := DT_in;
	esr_out[cnt].TS := TX;
	X6 := S6;
	cnt := cnt + 1;
	esr_flag := TRUE;
END_IF;
IF s7 <> X7  AND cnt < 4 THEN
	IF s7 THEN esr_out[cnt].typ := 11; ELSE 	esr_out[cnt].typ := 10; END_IF;
	esr_out[cnt].adress := a7;
	esr_out[cnt].DS := DT_in;
	esr_out[cnt].TS := TX;
	X7 := S7;
	cnt := cnt + 1;
	esr_flag := TRUE;
END_IF;
END_FUNCTION_BLOCK

(* POU ESR_MON_R4, ST *)
FUNCTION_BLOCK ESR_MON_R4
VAR_INPUT
	R0, R1, R2, R3 : REAL;
	DT_in : DT;
END_VAR
VAR_INPUT CONSTANT
	a0, a1, a2, a3 : STRING(10);
	s0, s1, s2, s3 : REAL;
END_VAR
VAR_OUTPUT
	ESR_Out: ARRAY [0..3] OF esr_data;
	ESR_Flag : BOOL;
END_VAR
VAR
	x0, x1, x2, x3 : REAL;
	tx: TIME;
	cnt : INT;
END_VAR

(*
version 1.0	26 jan 2007
programmer 	hugo
tested by		tobias

ESR_mon_R4 monitores up to 4 Real inputs and reports changes with time stamd and adress label.
the module checks 4 inputs for a change of more than the specified sensitivity S and reports all changes with time and adress stamp to the output.

*)
(* read system timer *)
tx := TIME();
ESR_Flag := FALSE;
esr_out[3].typ := 0;
esr_out[2].typ := 0;
esr_out[1].typ := 0;
esr_out[0].typ := 0;
cnt := 0;

(* check if inputs have chaged and fill buffer *)
IF differ(R0,  X0, S0) THEN
	esr_out[cnt].adress := a0;
	esr_out[cnt].DS := DT_in;
	esr_out[cnt].TS := TX;
	esr_out[cnt].data[0] := REAL_TO_BYTE(R0);
	esr_out[cnt].data[1] := DWORD_TO_BYTE(SHR(REAL_TO_DWORD(R0),8));
	esr_out[cnt].data[2] := DWORD_TO_BYTE(SHR(REAL_TO_DWORD(R0),16));
	esr_out[cnt].data[3] := DWORD_TO_BYTE(SHR(REAL_TO_DWORD(R0),24));
	X0 := R0;
	cnt := cnt + 1;
	esr_flag := TRUE;
END_IF;
IF differ(R1,  X1, S1) THEN
	esr_out[cnt].adress := a1;
	esr_out[cnt].DS := DT_in;
	esr_out[cnt].TS := TX;
	esr_out[cnt].data[0] := REAL_TO_BYTE(R1);
	esr_out[cnt].data[1] := DWORD_TO_BYTE(SHR(REAL_TO_DWORD(R1),8));
	esr_out[cnt].data[2] := DWORD_TO_BYTE(SHR(REAL_TO_DWORD(R1),16));
	esr_out[cnt].data[3] := DWORD_TO_BYTE(SHR(REAL_TO_DWORD(R1),24));
	X1 := R1;
	cnt := cnt + 1;
	esr_flag := TRUE;
END_IF;
IF differ(R2,  X2, S2) THEN
	esr_out[cnt].adress := a2;
	esr_out[cnt].DS := DT_in;
	esr_out[cnt].TS := TX;
	esr_out[cnt].data[0] := REAL_TO_BYTE(R2);
	esr_out[cnt].data[1] := DWORD_TO_BYTE(SHR(REAL_TO_DWORD(R2),8));
	esr_out[cnt].data[2] := DWORD_TO_BYTE(SHR(REAL_TO_DWORD(R2),16));
	esr_out[cnt].data[3] := DWORD_TO_BYTE(SHR(REAL_TO_DWORD(R2),24));
	X2 := R2;
	cnt := cnt + 1;
	esr_flag := TRUE;
END_IF;
IF differ(R3,  X3, S3) THEN
	esr_out[cnt].adress := a3;
	esr_out[cnt].DS := DT_in;
	esr_out[cnt].TS := TX;
	esr_out[cnt].data[0] := REAL_TO_BYTE(R3);
	esr_out[cnt].data[1] := DWORD_TO_BYTE(SHR(REAL_TO_DWORD(R3),8));
	esr_out[cnt].data[2] := DWORD_TO_BYTE(SHR(REAL_TO_DWORD(R3),16));
	esr_out[cnt].data[3] := DWORD_TO_BYTE(SHR(REAL_TO_DWORD(R3),24));
	X3 := R3;
	cnt := cnt + 1;
	esr_flag := TRUE;
END_IF;
END_FUNCTION_BLOCK

(* POU ESR_MON_X8, ST *)
FUNCTION_BLOCK ESR_MON_X8
VAR_INPUT
	s0, s1, s2, s3, s4, s5, s6, s7 : BYTE;
	DT_in : DT;
	Mode : BYTE := 3;
END_VAR
VAR_INPUT CONSTANT
	a0, a1, a2, a3, a4, a5, a6, a7 : STRING(10);
END_VAR
VAR_OUTPUT
	ESR_Out: ARRAY [0..3] OF esr_data;
	ESR_Flag : BOOL;
END_VAR
VAR
	x0, x1, x2, x3, x4, x5, x6, x7 : BYTE;
	tx: TIME;
	cnt : INT;
END_VAR

(*
version 1.0	26 jan 2007
programmer 	hugo
tested by		tobias

ESR_MON_X8 is a status and error collector.
the module checks 8 status inputs for a change and reports up to 4 input changes with time and adress stamp to the output.
the mode can be 
1 for error only
2 for error and status
3 for error, status and debug
the adress label of the 8 inputs can be configured individually.
*)
(* read system timer *)
tx := TIME();
ESR_Flag := FALSE;
esr_out[3].typ := 0;
esr_out[2].typ := 0;
esr_out[1].typ := 0;
esr_out[0].typ := 0;
cnt := 0;

(* check if inputs have chaged and fill buffer *)
IF s0 <> X0 AND ((s0 < 100) OR (S0 > 99 AND S0 < 200 AND mode >= 2) OR (S0 > 199 AND mode = 3)) THEN
	esr_out[cnt] := status_to_ESR(s0, a0, DT_in, TX);
	X0 := S0;
	cnt := cnt + 1;
	esr_flag := TRUE;
END_IF;
IF s1 <> X1 AND ((s1 < 100) OR (S1 > 99 AND S1 < 200 AND mode >= 2) OR (S1 > 199 AND mode = 3)) THEN
	esr_out[cnt] := status_to_ESR(s1, a1, DT_in, TX);
	X1 := S1;
	cnt := cnt + 1;
	esr_flag := TRUE;
END_IF;
IF s2 <> X2 AND ((s2 < 100) OR (S2 > 99 AND S2 < 200 AND mode >= 2) OR (S2 > 199 AND mode = 3)) THEN
	esr_out[cnt] := status_to_ESR(s2, a2, DT_in, TX);
	X2 := S2;
	cnt := cnt + 1;
	esr_flag := TRUE;
END_IF;
IF s3 <> X3 AND ((s3 < 100) OR (S3 > 99 AND S3 < 200 AND mode >= 2) OR (S3 > 199 AND mode = 3)) THEN
	esr_out[cnt] := status_to_ESR(s3, a3, DT_in, TX);
	X3 := S3;
	cnt := cnt + 1;
	esr_flag := TRUE;
END_IF;
IF cnt < 4 AND s4 <> X4 AND ((s4 < 100) OR (S4 > 99 AND S4 < 200 AND mode >= 2) OR (S4 > 199 AND mode = 3)) THEN
	esr_out[cnt] := status_to_ESR(s4, a4, DT_in, TX);
	X4 := S4;
	cnt := cnt + 1;
	esr_flag := TRUE;
END_IF;
IF cnt < 4 AND s5 <> X5 AND ((s5 < 100) OR (S5 > 99 AND S5 < 200 AND mode >= 2) OR (S5 > 199 AND mode = 3)) THEN
	esr_out[cnt] := status_to_ESR(s5, a5, DT_in, TX);
	X5 := S5;
	cnt := cnt + 1;
	esr_flag := TRUE;
END_IF;
IF cnt < 4 AND s6 <> X6 AND ((s6 < 100) OR (S6 > 99 AND S6 < 200 AND mode >= 2) OR (S6 > 199 AND mode = 3)) THEN
	esr_out[cnt] := status_to_ESR(s6, a6, DT_in, TX);
	X6 := S6;
	cnt := cnt + 1;
	esr_flag := TRUE;
END_IF;
IF cnt < 4 AND s7 <> X7 AND ((s7 < 100) OR (S7 > 99 AND S7 < 200 AND mode >= 2) OR (S7 > 199 AND mode = 3)) THEN
	esr_out[cnt] := status_to_ESR(s7, a7, DT_in, TX);
	X7 := S7;
	cnt := cnt + 1;
	esr_flag := TRUE;
END_IF;
END_FUNCTION_BLOCK

(* POU status_to_ESR, ST *)
FUNCTION status_to_ESR : esr_data
VAR_INPUT
	status : BYTE;
	adress : STRING(10);
	DT_in : DT;
	TS : TIME;
END_VAR
VAR
END_VAR

(*
version 1.0	6 oct 2006
programmer 	hugo
tested by		tobias

status_to_esr creates esr data from a status byte.

*)
IF status < 100 THEN
	status_to_ESR.typ := 1;
ELSIF status < 200 THEN
	status_to_ESR.typ := 2;
ELSE
	status_to_ESR.typ := 3;
END_IF;
status_to_ESR.adress:= adress;
status_to_ESR.DS := DT_in;
status_to_ESR.TS := TS;
status_to_ESR.data[0] := status;
END_FUNCTION

(* POU exec, ST *)
FUNCTION exec : STRING
VAR_INPUT
	str : STRING;
END_VAR
VAR
	pos: INT;
	R1: REAL;
	R2: REAL;
	operator: STRING;
END_VAR

(*
version 1.1	6 feb 2007
programmer 	hugo
tested by		tobias

exec executes a mathematical term and returns the result as a string
the term can only be a simple term without brackets and only one operator
allowed operastors are: (+, -, *, /, ^, sqrt, sin, cos, tan).

*)
(* extract both numbers and operator *)
exec := uppercase(trim(str));

pos := findB_nonum(exec);
IF pos > 1 THEN R1 := STRING_TO_REAL(exec); END_IF;
R2 := STRING_TO_REAL(RIGHT(exec,LEN(exec)-pos));
exec := LEFT(exec,pos);
pos := findB_Num(exec);
operator := RIGHT(exec,LEN(exec) - pos);
IF operator = '' AND LEN(str) = 0 THEN
	exec := '';
	RETURN;
ELSIF operator = '' THEN
	exec := str;
	RETURN;
END_IF;
IF operator = '^' THEN
	exec := REAL_TO_STRING(EXPT(R1, R2));
ELSIF operator = 'SQRT' THEN
	exec := REAL_TO_STRING(SQRT(R2));
ELSIF operator = 'SIN' THEN
	exec := REAL_TO_STRING(SIN(r2));
ELSIF operator = 'COS' THEN
	exec := REAL_TO_STRING(COS(r2));
ELSIF operator = 'TAN' THEN
	exec := REAL_TO_STRING(TAN(R2));
ELSIF operator = '*' THEN
	exec := REAL_TO_STRING(R1 * R2);
ELSIF operator = '/' THEN
	IF R2 <> 0 THEN exec := REAL_TO_STRING(R1 / R2); ELSE exec := 'ERROR'; END_IF;
ELSIF operator = '+' THEN
	exec := REAL_TO_STRING(r1 + r2);
ELSIF operator = '-' THEN
	exec := REAL_TO_STRING(r1 - r2);
ELSE
	exec := 'ERROR';
END_IF;


(* revision history

hm 6.feb 2007	rev 1.1
	cos has to be written in uppercase
	divide by 0 will return an error
     
*)
END_FUNCTION

(* POU uppercase, ST *)
FUNCTION uppercase : STRING
VAR_INPUT
	str : STRING;
END_VAR
VAR
	PT : POINTER TO BYTE;
	pos: INT;
END_VAR

(*
version 1.0	6 oct 2006
programmer 	hugo
tested by		tobias

uppercase returns str while all letters a..z are converted to uppercase

*)
PT := ADR(uppercase);
uppercase := str;
FOR pos := 1 TO LEN(str) DO
	IF PT^ > 96 AND PT^ < 123 THEN PT^ := PT^ - 32; END_IF;
	PT := PT + 1;
END_FOR;
END_FUNCTION

(* POU trim, ST *)
FUNCTION trim : STRING
VAR_INPUT
	str : STRING;
END_VAR
VAR
	pos: INT;
END_VAR

(*
version 1.0	6 oct 2006
programmer 	hugo
tested by		tobias

the function deletes all blanks within a string.

*)
trim := str;
REPEAT
	pos := FIND(trim,' ');
	trim := REPLACE(trim,'',1,pos);
UNTIL pos = 0	END_REPEAT;
END_FUNCTION

